# B&R Automation Studio project NAEUL004C00R13L518F00 (part 40)

### Buffer1.var - not listed in the package file held
```iecst
(*2019-06-07*)
(**)
(*Action & State & Status*)
VAR
	p_Buffer1Stat : UDINT;
	p_Buffer1Status : UDINT;
	p_Buffer1StatTxt : UDINT;
END_VAR
(**)
(*Alarm*)
VAR
	p_Buffer1AlmData : UDINT;
END_VAR
(**)
(*Output*)
VAR
	p_Buffer1NxtLoadSlt : UDINT;
	p_Buffer1NxtUnloadSlt : UDINT;
	p_Buffer1CoolBrdAny : UDINT;
	p_Buffer1CoolBrdGd : UDINT;
	p_Buffer1CoolBrdBad : UDINT;
	p_Buffer1CoolNotRdy : UDINT;
	p_Buffer1Bffr : UDINT;
	p_Buffer1DispBffr : UDINT;
	p_Buffer1BffrStat : UDINT;
	p_Buffer1BrdUnloadStat : UDINT;
	p_Buffer1FileNotFound : UDINT;
	p_Buffer1CoolFanCtrl : UDINT;
	p_Buffer1MagPresent : UDINT;
	p_Buffer1MagPresentTm : UDINT;
	p_Buffer1NewProduct : UDINT;
	p_Buffer1LastProductUnload : UDINT;
	p_Buffer1LastProductLeftInBffr : UDINT;
	p_Buffer1ParamDiff : UDINT;
	p_Buffer1MagRemoved : UDINT;
	p_Buffer1FIFOOld : UDINT;
	p_Buffer1SlotNo : UDINT;
END_VAR
```

### Buffer2.var - not listed in the package file held
```iecst
(*2019-03-25*)
(**)
(*Action & State & Status*)
VAR
	p_Buffer2Stat : UDINT;
	p_Buffer2Status : UDINT;
	p_Buffer2StatTxt : UDINT;
END_VAR
(**)
(*Alarm*)
VAR
	p_Buffer2AlmData : UDINT;
END_VAR
(**)
(*Output*)
VAR
	p_Buffer2NxtLoadSlt : UDINT;
	p_Buffer2NxtUnloadSlt : UDINT;
	p_Buffer2CoolBrdAny : UDINT;
	p_Buffer2CoolBrdGd : UDINT;
	p_Buffer2CoolBrdBad : UDINT;
	p_Buffer2CoolNotRdy : UDINT;
	p_Buffer2Bffr : UDINT;
	p_Buffer2DispBffr : UDINT;
	p_Buffer2BffrStat : UDINT;
	p_Buffer2BrdUnloadStat : UDINT;
	p_Buffer2FileNotFound : UDINT;
	p_Buffer2CoolFanCtrl : UDINT;
	p_Buffer2MagPresent : UDINT;
	p_Buffer2MagPresentTm : UDINT;
	p_Buffer2NewProduct : UDINT;
	p_Buffer2LastProductUnload : UDINT;
	p_Buffer2LastProductLeftInBffr : UDINT;
	p_Buffer2ParamDiff : UDINT;
	p_Buffer2MagRemoved : UDINT;
	p_Buffer2FIFOOld : UDINT;
	p_Buffer2SlotNo : UDINT;
END_VAR
```

### Buffer3.var - not listed in the package file held
```iecst
(*2019-03-25*)
(**)
(*Action & State & Status*)
VAR
	p_Buffer3Stat : UDINT;
	p_Buffer3Status : UDINT;
	p_Buffer3StatTxt : UDINT;
END_VAR
(**)
(*Alarm*)
VAR
	p_Buffer3AlmData : UDINT;
END_VAR
(**)
(*Output*)
VAR
	p_Buffer3NxtLoadSlt : UDINT;
	p_Buffer3NxtUnloadSlt : UDINT;
	p_Buffer3CoolBrdAny : UDINT;
	p_Buffer3CoolBrdGd : UDINT;
	p_Buffer3CoolBrdBad : UDINT;
	p_Buffer3CoolNotRdy : UDINT;
	p_Buffer3Bffr : UDINT;
	p_Buffer3DispBffr : UDINT;
	p_Buffer3BffrStat : UDINT;
	p_Buffer3BrdUnloadStat : UDINT;
	p_Buffer3FileNotFound : UDINT;
	p_Buffer3CoolFanCtrl : UDINT;
	p_Buffer3MagPresent : UDINT;
	p_Buffer3MagPresentTm : UDINT;
	p_Buffer3NewProduct : UDINT;
	p_Buffer3LastProductUnload : UDINT;
	p_Buffer3LastProductLeftInBffr : UDINT;
	p_Buffer3ParamDiff : UDINT;
	p_Buffer3MagRemoved : UDINT;
	p_Buffer3FIFOOld : UDINT;
	p_Buffer3SlotNo : UDINT;
END_VAR
```

### BufferMagA.var - not listed in the package file held
```iecst
(*2019-01-30*)
(**)
(*Action & State & Status*)
(**)
(*Alarm*)
(**)
(*Output*)
VAR
	p_BufferMagABffrMtySlt : UDINT;
END_VAR
```

### BufferMagB.var - not listed in the package file held
```iecst
(*2019-01-30*)
(**)
(*Action & State & Status*)
(**)
(*Alarm*)
(**)
(*Output*)
VAR
	p_BufferMagBBffrMtySlt : UDINT;
END_VAR
```

### SMEMA.typ - Do Not Change!!!
```iecst
(*2018-12-13*)
(**)
(*Action*)

TYPE
	eSMEMAAction :
		(
		SMEMAActIdle,
		SMEMAActRun,
		SMEMAActSetSig,
		SMEMAActSetStatSig,
		SMEMAActRstSig,
		SMEMAActRstStatSig,
		SMEMAActSetAllSig,
		SMEMAActRstAllSig
		);
END_TYPE

(**)

TYPE
	tySMEMAParam : 	STRUCT
		eSelection : eSMEMASelection;
		bStatSigSetGd : BOOL;
	END_STRUCT;
	eSMEMASelection :
		(
		SMEMASelStandard,
		SMEMASelIPC9851,
		SMEMASelIPC9851Ext
		);
	tyUSSMEMA : 	STRUCT
		In : tyUSSMEMAIn1;
		Out : tyUSSMEMAAOut1;
	END_STRUCT;
	tyUSSMEMAIn1 : 	STRUCT
		eAct : eSMEMAAction := SMEMAActIdle; (*USSMEMA Act*)
		udiRstErr : UDINT := 0; (*Reset Error*)
		bPrep : BOOL := TRUE; (*Project Preparation*)
		bEn : BOOL := TRUE; (*Enable*)
		bDis : BOOL := FALSE; (*Disable*)
		bRdyRcv : BOOL := TRUE; (*Ready Receive Signal*)
		bLeftSen : BOOL := FALSE; (*Left Sensor*)
		bRightSen : BOOL := FALSE; (*Right Sensor*)
		bComplSigOn : BOOL := FALSE; (*Complete Signal is On*)
		bUBA : BOOL := FALSE; (*Upstream is Available Signal*)
		bUBAStat : BOOL := FALSE; (*Upstream is Available Signal's State*)
		bTimerEnSen : BOOL; (*Timer Enable Sensor*)
		bTimerEnSenEdge : BOOL; (*Timer Enable Sensor Edge*)
		bVirtualEn : BOOL; (*Virtual Mode Enable*)
		bUBAVirtual : BOOL; (*Upstream Available Vritual Signal*)
		bUBAStatVirtual : BOOL; (*Upstream Available Vritual Signal's State*)
		tyParam : tySMEMAParam; (*SMEMA Parameter*)
		diTransferInTO : DINT := 20000; (*Transfer Out Timer On*)
		bDirLToR : BOOL := FALSE; (*Direction Left to Right*)
		tRstDlyTm : TIME := T#500ms; (*Reset Delay Timer*)
		tSigInChkTm : TIME := T#100ms; (*Signal In Check Timer*)
		sProgNm : STRING[15] := 'USSMEMA'; (*Program's Name*)
		bNtSettingsLoadDone : BOOL := TRUE; (*Nutek Parameter Settings Loading is Done*)
	END_STRUCT;
	tyUSSMEMAAOut1 : 	STRUCT
		eStat : eBufferAction := BufferActIdle; (*Hardware Info's State*)
		eStatus : eFBStatus := Idle; (*Hardware Info's Status*)
		sStatTxt : STRING[200] := ''; (*Hardware Info's State in Text*)
		tyAlmData : tyAlmDat; (*Alarm Data*)
		bUSRdy : BOOL := FALSE; (*Upstream is Ready*)
		bUSGdBrdRdy : BOOL := FALSE; (*Upstream Good Board is Ready*)
		bDSRdy : BOOL := FALSE; (*Downstream is Ready*)
		bTransporting : BOOL := FALSE; (*Is Transporting*)
		bConvStart : BOOL := FALSE; (*Converyor Starts*)
		bConvStop : BOOL := FALSE; (*Conveyor Stop*)
		bUSB : BOOL := FALSE; (*Upstream Busy Signal*)
		bTimer : BOOL; (*Timer is On*)
		bVirtual : BOOL; (*Virtual Mode is On*)
	END_STRUCT;
	tyDSSMEMA : 	STRUCT
		In : tyDSSMEMAIn1;
		Out : tyDSSMEMAOut1;
	END_STRUCT;
	tyDSSMEMAIn1 : 	STRUCT
		eAct : eSMEMAAction := SMEMAActIdle; (*DSSMEMA Act*)
		udiRstErr : UDINT := 0; (*Reset Error*)
		bPrep : BOOL := TRUE; (*Project Preparation*)
		bEn : BOOL := TRUE; (*Enable*)
		bDis : BOOL := FALSE; (*Disable*)
		bGdBrd : BOOL := TRUE; (*Have Good Board*)
		bRdySend : BOOL := TRUE; (*Ready Send Signal*)
		bLeftSen : BOOL := FALSE; (*Left Sensor*)
		bRightSen : BOOL := FALSE; (*Right Sensor*)
		bClrSen : BOOL;
		bComplSigOn : BOOL := FALSE; (*Complete Signal is On*)
		bDSB : BOOL := FALSE; (*Downstream Busy Signal*)
		bTimerEnSen : BOOL; (*Timer Enable Sensor*)
		bTimerEnSenEdge : BOOL; (*Timer Enable Sensor Edge*)
		bVirtualEn : BOOL; (*Virtual Mode Enable*)
		bDSBVirtual : BOOL; (*Downstream Busy Signal*)
		tyParam : tySMEMAParam; (*SMEMA Parameter*)
		diTransferOutTO : DINT := 20000;
		bDirLToR : BOOL := FALSE; (*Direction Left to Right*)
		tRstDlyTm : TIME := T#500ms; (*Reset Delay Timer*)
		tSigInChkTm : TIME := T#100ms; (*Signal In Check Timer*)
		sProgNm : STRING[15] := 'USSMEMA'; (*Program's Name*)
		bNtSettingsLoadDone : BOOL := TRUE; (*Nutek Parameter Settings Loading is Done*)
	END_STRUCT;
	tyDSSMEMAOut1 : 	STRUCT
		eStat : eSMEMAAction := SMEMAActIdle; (*DSSMEMA's State*)
		eStatus : eFBStatus := Idle; (*DSSMEMA's Status*)
		sStatTxt : STRING[200] := ''; (*DSSMEMA's State in Text*)
		tyAlmData : tyAlmDat; (*Alarm Data*)
		bUSRdy : BOOL := FALSE; (*Upstream is Ready*)
		bUSGdBrdRdy : BOOL := FALSE; (*Upstream Good Board is Ready*)
		bDSRdy : BOOL := FALSE; (*Downstream is Ready*)
		bTransporting : BOOL := FALSE; (*Is Transporting*)
		bConvStart : BOOL := FALSE; (*Conveyor Start*)
		bConvStop : BOOL := FALSE; (*Conveyor Stop*)
		bDBA : BOOL := FALSE; (*Downstream Available Signal*)
		bDBAStat : BOOL := FALSE; (*Downstream Avaialble Signal's State*)
		bTimer : BOOL; (*Timer is On*)
		bVirtual : BOOL; (*Virtual Mode is Mode*)
	END_STRUCT;
END_TYPE
```

### USSMEMAA.var - Change By Project
```iecst
(**)
VAR
	g_tyUSSMEMAA : tyUSSMEMAAOut1; (*Upstream SMEMA*)
END_VAR
```

### Program Logical/SMEMA/USSMEMAA (IEC) - 1.00.0 - NtSMEMA v5.00.0

#### InputRef_Link.var
```iecst
(*2019-04-09*)
(**)
(*External Data*)
VAR
	p_bLinkOpsRun : REFERENCE TO BOOL;
END_VAR
(**)
VAR
	p_eLinkConvDir : REFERENCE TO eConvDir;
	p_eLinkOpsTravLifPosGo : REFERENCE TO eTravLifULPos;
	p_bLinkConvHvBrd : REFERENCE TO BOOL;
	p_bLinkNtParamUSWidthChkPrep : REFERENCE TO BOOL;
	p_bLinkMcParamUSWidthChkEn : REFERENCE TO BOOL;
	p_bLinkDIUSWidthChkSen : REFERENCE TO BOOL;
END_VAR
```

#### Act_Alarm.st
```iecst
(** 2019-03-25 **)
ACTION Act_Alarm:
	//Reset Error
	IF tylocalUSSMEMA.In.udiRstErr <> udiRstErrOld THEN
		bRstErr			:= TRUE;
		udiRstErrOld	:= tylocalUSSMEMA.In.udiRstErr;
	ELSE
		bRstErr			:= FALSE;
	END_IF

	//Error State
	IF (tylocalUSSMEMA.Out.eStatus = Error) AND bRstErr THEN
		tylocalUSSMEMA.In.eAct		:= SMEMAActIdle;
		tylocalUSSMEMA.Out.eStat	:= SMEMAActIdle;
	END_IF

	//Error Link To HMI
	IF EDGEPOS(tylocalUSSMEMA.Out.eStatus = Error) THEN

		tylocalUSSMEMA.Out.tyAlmData.udiCode		:= udiStatus;
		tylocalUSSMEMA.Out.tyAlmData.eSeverity		:= AlmSeverityError;
		tylocalUSSMEMA.Out.tyAlmData.udiRunTime		:= tylocalUSSMEMA.Out.tyAlmData.udiRunTime + 1;
		tylocalUSSMEMA.Out.tyAlmData.bAlm			:= TRUE;
		tylocalUSSMEMA.Out.tyAlmData.udiModuleNum	:= udiModuleNum;
		g_tyAlmProgNm.sUSSMEMAProgNm				:= tylocalUSSMEMA.In.sProgNm;

	ELSIF bRstErr AND (tylocalUSSMEMA.Out.tyAlmData.udiCode <> 0) THEN

		tylocalUSSMEMA.Out.tyAlmData.udiCode	:= 0;
		tylocalUSSMEMA.Out.tyAlmData.eSeverity	:= AlmSeverityNA;
		tylocalUSSMEMA.Out.tyAlmData.bAlm		:= FALSE;

		tylocalUSSMEMA.Out.sStatTxt	:= a_sStatText[tylocalUSSMEMA.Out.eStat];

	END_IF

END_ACTION
```

#### Act_InitGlobal.st
```iecst
(** 2019-04-09 **)
ACTION Act_InitGlobal:

	(* Always Change If Project Change *)

	//Pass Data To Link
	p_bLinkOpsRun ACCESS p_OpsRun;

	p_eLinkConvDir ACCESS p_NtParamProjConvDir;
	p_eLinkOpsTravLifPosGo ACCESS p_OpsTravLifULPosGo;
	p_bLinkConvHvBrd ACCESS p_PshrConvHvBrd;
	p_bLinkNtParamUSWidthChkPrep ACCESS p_NtParamUSWidthChkPrep;
	p_bLinkMcParamUSWidthChkEn ACCESS p_McParamUSWidthChkEn;
	p_bLinkDIUSWidthChkSen ACCESS p_DIUSWidthChkSen;

	//Pass Data To Internal Use
	p_udiRstErr ACCESS p_RstErrReset;
	p_bManual ACCESS p_UIMnlMod;
	p_tyParam ACCESS p_McParamUSSMEMAAParam;
	p_diTransferInTO ACCESS p_McParamTranInErrDlyTm;
	p_bLeftSen ACCESS p_DIConvLftSen;
	p_bRightSen ACCESS p_DIConvRgtSen;
	p_bUBA ACCESS p_DIUBAA;
	p_bUBAStat ACCESS p_DIUBAAStat;
	p_bVirtualEn ACCESS p_UIVSMEMAUSAEn;
	p_bUBAVirtual ACCESS p_UIVSMEMAUBAA;
	p_bUBAStatVirtual ACCESS p_UIVSMEMAUBAAStat;
	p_tRstDlyTm ACCESS p_NtParamUSSMEMAARstDlyTm;
	p_tSigInChkTm ACCESS p_NtParamUSSMEMAASigInChkTm;
	p_sProgNm ACCESS p_NtParamUSSMEMAAProgNm;
	p_bNtSettingsLoadDone ACCESS p_StartupNtSettingsLoadDone;
	p_bLinkOpsTravLifULUSComm ACCESS p_OpsTravLifULUSComm;
	(* Always Change If Project Change *)

END_ACTION
```

#### Act_InputConfig.st
```iecst
(** 2019-04-09 **)
ACTION Act_InputConfig:

	(* Always Change If Project Change *)

	//Pass Data To Link
	tylocalUSSMEMA.In.udiRstErr := g_tyRstErr.bReset;
	tylocalUSSMEMA.In.tyParam := g_tyMcParamCurr.tyUSCommASMEMA;
	tylocalUSSMEMA.In.diTransferInTO := g_tyMcParamCurr.diTranInErrDlyTmInMS;
	tylocalUSSMEMA.In.bLeftSen := g_tyDInput.bConvLftSen;
	tylocalUSSMEMA.In.bRightSen := g_tyDInput.bConvRgtSen;
	tylocalUSSMEMA.In.bUBA := g_tyDInput.bUBAA;
	tylocalUSSMEMA.In.bUBAStat := g_tyDInput.bUBAAStat;
	tylocalUSSMEMA.In.bVirtualEn := g_tyUIOut.bVSMEMAUSAEn;
	tylocalUSSMEMA.In.bUBAVirtual := g_tyUIOut.bVSMEMAUBAA;
	tylocalUSSMEMA.In.bUBAStatVirtual := g_tyUIOut.bVSMEMAUBAAStat;
	tylocalUSSMEMA.In.tRstDlyTm := g_tyNtParamCurr.tUSSMEMAARstDlyTm;
	tylocalUSSMEMA.In.tSigInChkTm := g_tyNtParamCurrt.tUSSMEMAASigInChkTm;
	tylocalUSSMEMA.In.sProgNm := g_tyNtParamCurr.sUSSMEMAAProgNm;

	//Ready Receive
	IF g_tyNtParamCurr.bUSWidthChkPrep AND g_tyMcParamCurr.bUSWidthChkEn THEN
		tylocalUSSMEMA.In.bRdyRcv	:= (g_tyDInput.bnput.bUSWidthChkSen = TRUE) AND (g_tyPshrConv.bHvBrd = FALSE) AND (g_tyOpsTravLifUL.eTravLifULPosGo = TravLifULPosUS1);
	ELSE
		tylocalUSSMEMA.In.bRdyRcv	:= (g_tyPshrConv.bHvBrd = FALSE) AND (g_tyOpsTravLifUL.eTravLifULPosGo = TravLifULPosUS1) AND g_tyOps.bTravLifULUSComm;
	END_IF

	//Receive Complete Signal
	//	tylocalUSSMEMA.In.bComplSigOn	:= tylocalUSSMEMA.In.bLeftSen = FALSE;
	IF EDGENEG(tylocalUSSMEMA.In.bLeftSen) THEN
		tylocalUSSMEMA.In.bComplSigOn	:= TRUE;
	END_IF

	IF tylocalUSSMEMA.Out.eStat <> SMEMAActRun THEN
		tylocalUSSMEMA.In.bComplSigOn	:= FALSE;
	END_IF

	//Direction
	tylocalUSSMEMA.In.bDirLToR	:= g_tyNtParamCurr.eProjConvDir = ConvDirLToR OR g_tyNtParamCurr.eProjConvDir = ConvDirRToL;

	IF g_tyOps.bRun = TRUE THEN
		tylocalUSSMEMA.In.eAct := g_tyOpsTravLifUL.eUSSMEMAAct1;
	ELSIF g_tyUIOut.Out.bManualMod = TRUE THEN
		tylocalUSSMEMA.In.eAct := g_tyUIOut.eMnlAct.eUSSMEMAAAct;
	ELSE
		tylocalUSSMEMA.In.eAct ACCESS ADR(eAct);
	END_IF

END_ACTION
```

#### Act_Link.st
```iecst
(** 2019-03-29 **)
ACTION Act_Link:

	//Ready Receive
	IF p_bLinkNtParamUSWidthChkPrep AND p_bLinkMcParamUSWidthChkEn THEN
		p_bRdyRcv	:= (p_bLinkDIUSWidthChkSen = TRUE) AND (p_bLinkConvHvBrd = FALSE) AND (p_eLinkOpsTravLifPosGo = TravLifULPosUS1);
	ELSE
		p_bRdyRcv	:= (p_bLinkConvHvBrd = FALSE) AND (p_eLinkOpsTravLifPosGo = TravLifULPosUS1) AND p_bLinkOpsTravLifULUSComm;
	END_IF

	//Receive Complete Signal
//	p_bComplSigOn	:= p_bLeftSen = FALSE;
	IF EDGENEG(p_bLeftSen) THEN
		p_bComplSigOn	:= TRUE;
	END_IF

	IF eStat <> SMEMAActRun THEN
		p_bComplSigOn	:= FALSE;
	END_IF

	//Direction
	p_bDirLToR	:= p_eLinkConvDir = ConvDirLToR OR p_eLinkConvDir = ConvDirLToL;

END_ACTION
```

#### Act_LinkAction.st
```iecst
(** 2019-04-09 **)
ACTION Act_LinkAction:

	IF p_bLinkOpsRun = TRUE THEN
		p_eAct ACCESS p_OpsTravLifULUSSMEMAAct1;
	ELSIF p_bManual = TRUE THEN
		p_eAct ACCESS p_UIUSSMEMAAAct;
	ELSE
		p_eAct ACCESS ADR(eAct);
	END_IF

END_ACTION
```

#### Act_Main.st
```iecst
ACTION Act_Main:

	fbSMEMA_Std.tRstDlyTm 		:= tylocalUSSMEMA.In.tRstDlyTm;
	fbSMEMA_9851.tRstDlyTm  	:= tylocalUSSMEMA.In.tRstDlyTm;
	fbSigInChk.tSigInChkTm		:= tylocalUSSMEMA.In.tSigInChkTm;

	//Timer Running
	fbTimeTrig(CLK := tylocalUSSMEMA.In.bTimerEnSenEdge);

	IF tylocalUSSMEMA.Out.eStat = SMEMAActRun AND (tylocalUSSMEMA.In.bTimerEnSenEdge OR tylocalUSSMEMA.In.bTimerEnSen) THEN
		IF fbTimeTrig.Q = TRUE OR tylocalUSSMEMA.In.bTimerEnSen THEN
			fbTimerDlyTm.IN	:= TRUE;
		END_IF
	ELSE
		fbTimerDlyTm.IN	:= FALSE;
	END_IF

	IF tylocalUSSMEMA.Out.bConvStart = FALSE AND tylocalUSSMEMA.Out.bConvStop = FALSE THEN
		fbTimerDlyTm;

		IF fbTimerDlyTm.Q = TRUE AND tylocalUSSMEMA.Out.eStat = SMEMAActRun THEN
			tylocalUSSMEMA.Out.bTimer		:= TRUE;
			tylocalUSSMEMA.Out.bVirtual		:= FALSE;
		ELSIF tylocalUSSMEMA.In.bVirtualEn = TRUE THEN
			tylocalUSSMEMA.Out.bTimer		:= FALSE;
			tylocalUSSMEMA.Out.bVirtual		:= TRUE;
		ELSE
			tylocalUSSMEMA.Out.bTimer		:= FALSE;
			tylocalUSSMEMA.Out.bVirtual		:= FALSE;
		END_IF
	ELSE
		fbTimerDlyTm(IN := FALSE);
	END_IF

	IF tylocalUSSMEMA.Out.bTimer = TRUE THEN

		fbSigInChk.bNomSig			:= tylocalUSSMEMA.Out.bConvStart = FALSE AND tylocalUSSMEMA.Out.bConvStop = FALSE;
		fbSigInChk.bStatSig			:= FALSE;
		fbSigInChk.bStatSigSetGd	:= FALSE;

	ELSIF tylocalUSSMEMA.Out.bVirtual = TRUE THEN

		fbSigInChk.bNomSig	:= tylocalUSSMEMA.In.bUBAVirtual;

		IF tylocalUSSMEMA.In.tyParam.eSelection = SMEMASelIPC9851Ext THEN
			fbSigInChk.bStatSig			:= tylocalUSSMEMA.In.bUBAStatVirtual;
			fbSigInChk.bStatSigSetGd	:= tylocalUSSMEMA.In.tyParam.bStatSigSetGd;
		ELSE
			fbSigInChk.bStatSig			:= FALSE;
			fbSigInChk.bStatSigSetGd	:= FALSE;
		END_IF

	ELSE

		fbSigInChk.bNomSig	:= tylocalUSSMEMA.In.bUBA;

		IF tylocalUSSMEMA.In.tyParam.eSelection = SMEMASelIPC9851Ext THEN
			fbSigInChk.bStatSig			:= tylocalUSSMEMA.In.bUBAStat;
			fbSigInChk.bStatSigSetGd	:= tylocalUSSMEMA.In.tyParam.bStatSigSetGd;
		ELSE
			fbSigInChk.bStatSig			:= FALSE;
			fbSigInChk.bStatSigSetGd	:= FALSE;
		END_IF

	END_IF

	fbSigInChk;

	tylocalUSSMEMA.Out.bUSRdy		    := fbSigInChk.bSigInValid;
	tylocalUSSMEMA.Out.bUSGdBrdRdy   	:= fbSigInChk.bGdBrd;

	//Set p_eAct
	IF tylocalUSSMEMA.Out.eStatus = Idle OR tylocalUSSMEMA.Out.eStatus = Busy OR tylocalUSSMEMA.Out.eStatus = Done THEN
		tylocalUSSMEMA.Out.eStatus	:= tylocalUSSMEMA.In.eAct;
	END_IF

	//Transition State
	IF eStatOld <> tylocalUSSMEMA.Out.eStat THEN

		fbSMEMA_Std(bEn := FALSE);
		fbSMEMA_9851(bEn := FALSE);

		tylocalUSSMEMA.Out.bTransporting	:= FALSE;
		tylocalUSSMEMA.Out.bConvStart		:= FALSE;
		tylocalUSSMEMA.Out.bConvStop		:= FALSE;
		tylocalUSSMEMA.Out.bDSRdy			:= FALSE;

		IF eStatOld <> SMEMAActIdle
			AND eStatOld <> SMEMAActSetSig
			AND eStatOld <> SMEMAActSetStatSig
			AND eStatOld <> SMEMAActRstSig
			AND eStatOld <> SMEMAActRstStatSig
			AND eStatOld <> SMEMAActSetAllSig
			AND eStatOld <> SMEMAActRstAllSig THEN

			tylocalUSSMEMA.Out.bUSB	:= FALSE;

		END_IF

		tylocalUSSMEMA.Out.sStatTxt	:= a_sStatText[tylocalUSSMEMA.Out.eStat];

		eStatOld	:= tylocalUSSMEMA.Out.eStat;

		tylocalUSSMEMA.Out.eStatus		:= Busy;
	END_IF

	//Inlet Sensor & Outlet Sensor
	IF tylocalUSSMEMA.In.bDirLToR THEN
		bInletSen 	:= tylocalUSSMEMA.In.bLeftSen;
		bOutletSen  := tylocalUSSMEMA.In.bRightSen;
	ELSE
		bInletSen   := tylocalUSSMEMA.In.bRightSen;
		bOutletSen  := tylocalUSSMEMA.In.bLeftSen;
	END_IF

	//Main
	CASE tylocalUSSMEMA.Out.eStat OF

		SMEMAActIdle:

			IF EDGENEG(g_tyUIOut.bManualMod) THEN
				tylocalUSSMEMA.Out.bUSB	:= FALSE;
			END_IF

			tylocalUSSMEMA.Out.eStatus	:= Idle;

		SMEMAActRun:
			IF tylocalUSSMEMA.Out.eStatus = Idle OR tylocalUSSMEMA.Out.eStatus = Busy THEN

				tylocalUSSMEMA.Out.eStatus	:= Busy;

				IF tylocalUSSMEMA.In.tyParam.eSelection <> SMEMASelStandard THEN

					fbSMEMA_9851.bUSRdy			:= fbSigInChk.bSigInValid;
					fbSMEMA_9851.bRdyRcv		:= tylocalUSSMEMA.In.bRdyRcv;
					fbSMEMA_9851.bComplSigOn	:= tylocalUSSMEMA.In.bComplSigOn;
					fbSMEMA_9851.bInletSen		:= bInletSen;
					fbSMEMA_9851.bOutletSen		:= bOutletSen;

					fbSMEMA_9851.tTimeOut		:= DINT_TO_TIME(tylocalUSSMEMA.In.diTransferInTO);
					fbSMEMA_9851(bEn := TRUE);

					tylocalUSSMEMA.Out.bTransporting	:= fbSMEMA_9851.bTransporting;
					tylocalUSSMEMA.Out.bConvStart		:= fbSMEMA_9851.bConvStart;
					tylocalUSSMEMA.Out.bConvStop		:= fbSMEMA_9851.bConvStop;
					tylocalUSSMEMA.Out.bUSB				:= fbSMEMA_9851.bSigToUS AND (tylocalUSSMEMA.Out.bTimer = FALSE) AND (tylocalUSSMEMA.Out.bVirtual = FALSE);
					tylocalUSSMEMA.Out.bDSRdy			:= fbSMEMA_9851.bSigToUS;

					IF fbSMEMA_9851.udiStatus = 0 THEN
						tylocalUSSMEMA.Out.eStatus	:= Done;
					ELSIF fbSMEMA_9851.udiStatus < 65534 THEN
						tylocalUSSMEMA.Out.eStatus		:= Error;

						IF fbSMEMA_9851.udiStatus = 1200 THEN
							udiStatus	:= 2701;	//SMEMA 9851 Transport Time Out While Transporting
						ELSIF fbSMEMA_9851.udiStatus = 1201 THEN
							udiStatus	:= 2702;	//SMEMA 9851 Transport Time Out After Opposite Machine Transport Finished
						ELSIF fbSMEMA_9851.udiStatus = 1202 THEN
							udiStatus	:= 2703;	//SMEMA 9851 Transport Time Out After Current Machine Transport Finished
						ELSIF fbSMEMA_9851.udiStatus = 1203 THEN
							udiStatus	:= 2704;	//SMEMA 9851 Transport Time Out After Both Machine Transport Finished And Waiting Outlet Sensor
						ELSE
							udiStatus	:= fbSMEMA_9851.udiStatus;
						END_IF
					END_IF

				ELSE

					fbSMEMA_Std.bUSRdy		:= fbSigInChk.bSigInValid;
					fbSMEMA_Std.bRdyRcv		:= tylocalUSSMEMA.In.bRdyRcv;
					fbSMEMA_Std.bComplSigOn	:= tylocalUSSMEMA.In.bComplSigOn;
					fbSMEMA_Std.bInletSen	:= bInletSen;
					fbSMEMA_Std.bOutletSen	:= bOutletSen;
					fbSMEMA_Std.tTimeOut	:= DINT_TO_TIME(tylocalUSSMEMA.In.diTransferInTO);
					fbSMEMA_Std(bEn := TRUE);

					tylocalUSSMEMA.Out.bTransporting	:= fbSMEMA_Std.bTransporting;
					tylocalUSSMEMA.Out.bConvStart		:= fbSMEMA_Std.bConvStart;
					tylocalUSSMEMA.Out.bConvStop		:= fbSMEMA_Std.bConvStop;
					tylocalUSSMEMA.Out.bUSB				:= fbSMEMA_Std.bSigToUS AND (tylocalUSSMEMA.Out.bTimer = FALSE) AND (tylocalUSSMEMA.Out.bVirtual = FALSE);
					tylocalUSSMEMA.Out.bDSRdy			:= fbSMEMA_Std.bSigToUS;

					IF fbSMEMA_Std.udiStatus = 0 THEN
						tylocalUSSMEMA.Out.eStatus	:= Done;
					ELSIF fbSMEMA_Std.udiStatus < 65534 THEN
						tylocalUSSMEMA.Out.eStatus		:= Error;

						IF fbSMEMA_Std.udiStatus = 1200 THEN
							udiStatus	:= 2705;	//Standard SMEMA Transport Time Out While Transporting
						ELSIF fbSMEMA_Std.udiStatus = 1201 THEN
							udiStatus	:= 2706;	//Standard SMEMA Transport Time Out After Opposite Machine Transport Finished
						ELSIF fbSMEMA_Std.udiStatus = 1202 THEN
							udiStatus	:= 2707;	//Standard SMEMA Transport Time Out After Current Machine Transport Finished
						ELSIF fbSMEMA_Std.udiStatus = 1203 THEN
							udiStatus	:= 2708;	//Standard SMEMA Transport Time Out After Both Machine Transport Finished And Waiting Outlet Sensor
						ELSE
							udiStatus	:= fbSMEMA_Std.udiStatus;
						END_IF
					END_IF

				END_IF

			END_IF

		SMEMAActSetSig:
			IF tylocalUSSMEMA.Out.eStatus = Idle OR tylocalUSSMEMA.Out.eStatus = Busy THEN

				//Reset
				fbSMEMA_Std(bEn := FALSE);
				fbSMEMA_9851(bEn := FALSE);

				tylocalUSSMEMA.Out.bConvStart	:= FALSE;
				tylocalUSSMEMA.Out.bConvStop	:= FALSE;

				tylocalUSSMEMA.Out.bUSB		:= TRUE;
				tylocalUSSMEMA.Out.eStatus	:= Done;

			END_IF

		SMEMAActSetStatSig:
			IF tylocalUSSMEMA.Out.eStatus = Idle OR tylocalUSSMEMA.Out.eStatus = Busy THEN

				//Reset
				fbSMEMA_Std(bEn := FALSE);
				fbSMEMA_9851(bEn := FALSE);

				tylocalUSSMEMA.Out.bConvStart	:= FALSE;
				tylocalUSSMEMA.Out.bConvStop	:= FALSE;

				tylocalUSSMEMA.Out.eStatus	:= Done;

			END_IF

		SMEMAActRstSig:
			IF tylocalUSSMEMA.Out.eStatus = Idle OR tylocalUSSMEMA.Out.eStatus = Busy THEN

				//Reset
				fbSMEMA_Std(bEn := FALSE);
				fbSMEMA_9851(bEn := FALSE);

				tylocalUSSMEMA.Out.bConvStart	:= FALSE;
				tylocalUSSMEMA.Out.bConvStop	:= FALSE;

				tylocalUSSMEMA.Out.bUSB	:= FALSE;
				tylocalUSSMEMA.Out.eStatus	:= Done;

			END_IF

		SMEMAActRstStatSig:
			IF tylocalUSSMEMA.Out.eStatus = Idle OR tylocalUSSMEMA.Out.eStatus = Busy THEN

				//Reset
				fbSMEMA_Std(bEn := FALSE);
				fbSMEMA_9851(bEn := FALSE);

				tylocalUSSMEMA.Out.bConvStart	:= FALSE;
				tylocalUSSMEMA.Out.bConvStop	:= FALSE;

				tylocalUSSMEMA.Out.eStatus	:= Done;

			END_IF

		SMEMAActSetAllSig:
			IF tylocalUSSMEMA.Out.eStatus = Idle OR tylocalUSSMEMA.Out.eStatus = Busy THEN

				//Reset
				fbSMEMA_Std(bEn := FALSE);
				fbSMEMA_9851(bEn := FALSE);

				tylocalUSSMEMA.Out.bConvStart	:= FALSE;
				tylocalUSSMEMA.Out.bConvStop	:= FALSE;

				tylocalUSSMEMA.Out.bUSB	:= TRUE;
				tylocalUSSMEMA.Out.eStatus	:= Done;

			END_IF

		SMEMAActRstAllSig:
			IF tylocalUSSMEMA.Out.eStatus = Idle OR tylocalUSSMEMA.Out.eStatus = Busy THEN

				//Reset
				fbSMEMA_Std(bEn := FALSE);
				fbSMEMA_9851(bEn := FALSE);

				tylocalUSSMEMA.Out.bConvStart	:= FALSE;
				tylocalUSSMEMA.Out.bConvStop	:= FALSE;

				tylocalUSSMEMA.Out.bUSB	:= FALSE;
				tylocalUSSMEMA.Out.eStatus	:= Done;

			END_IF

	END_CASE

END_ACTION
```

#### Act_OutputConfig.st
```iecst
(** 2019-03-25 **)
ACTION Act_OutputConfig:

	g_tyUSSMEMAA := tylocalUSSMEMA.Out; // Change the Global Naming According to the Physical Hardware Module

END_ACTION
```

#### Init.st
```iecst
(** 2019-03-25 **)
PROGRAM _INIT

	(* Always Change If Project Change *)

	//Pass Address To Global Address For External Use
	//Action, State & Status
	p_USSMEMAAStat		:= ADR(eStat);
	p_USSMEMAAStatus		:= ADR(eStatus);
	p_USSMEMAAStatTxt	:= ADR(sStatTxt);

	//Alarm
	p_USSMEMAAAlmData	:= ADR(tyAlmData);

	//Output
	p_USSMEMAAUSRdy			:= ADR(bUSRdy);
	p_USSMEMAAUSGdBrdRdy	:= ADR(bUSGdBrdRdy);
	p_USSMEMAADSRdy			:= ADR(bDSRdy);
	p_USSMEMAATransporting	:= ADR(bTransporting);
	p_USSMEMAAConvStart		:= ADR(bConvStart);
	p_USSMEMAAConvStop		:= ADR(bConvStop);
	p_USSMEMAAUSB			:= ADR(bUSB);
	p_USSMEMAATimer			:= ADR(bTimer);
	p_USSMEMAAVirtual		:= ADR(bVirtual);

	(* Always Change If Project Change *)

END_PROGRAM
```

### USSMEMAB.var - Change By Project
```iecst
VAR
	g_tyUSSMEMAB : tyUSSMEMAAOut1;
END_VAR
```

### Program Logical/SMEMA/USSMEMAB (IEC) - 1.00.0 - NtSMEMA v5.00.0

#### InputRef.var
```iecst
(*2019-03-25*)
(**)
(*General*)
VAR
	p_eAct : REFERENCE TO eSMEMAAction;
	p_udiRstErr : REFERENCE TO UDINT;
	p_bPrep : REFERENCE TO BOOL;
	p_bEn : REFERENCE TO BOOL;
	p_bDis : REFERENCE TO BOOL;
END_VAR
(**)
(*Configuration*)
VAR
	p_bManual : REFERENCE TO BOOL;
	p_tyParam : REFERENCE TO tySMEMAParam;
	p_diTransferInTO : REFERENCE TO DINT;
	p_bDirLToR : REFERENCE TO BOOL;
	p_bRdyRcv : REFERENCE TO BOOL;
END_VAR
(**)
(*Input*)
VAR
	p_bLeftSen : REFERENCE TO BOOL;
	p_bRightSen : REFERENCE TO BOOL;
	p_bComplSigOn : REFERENCE TO BOOL;
	p_bUBA : REFERENCE TO BOOL;
	p_bUBAStat : REFERENCE TO BOOL;
	p_bTimerEnSen : REFERENCE TO BOOL;
	p_bTimerEnSenEdge : REFERENCE TO BOOL;
	p_bVirtualEn : REFERENCE TO BOOL;
	p_bUBAVirtual : REFERENCE TO BOOL;
	p_bUBAStatVirtual : REFERENCE TO BOOL;
	p_tRstDlyTm : REFERENCE TO TIME;
	p_tSigInChkTm : REFERENCE TO TIME;
	p_sProgNm : REFERENCE TO STRING[15];
	p_bNtSettingsLoadDone : REFERENCE TO BOOL;
	p_bLinkOpsTravLifULUSComm : REFERENCE TO BOOL;
END_VAR
```

#### Act_InitGlobal.st
```iecst
(** 2019-04-09 **)
ACTION Act_InitGlobal:

	(* Always Change If Project Change *)

	//Pass Data To Link
	p_bLinkOpsRun ACCESS p_OpsRun;

	p_eLinkConvDir ACCESS p_NtParamProjConvDir;
	p_eLinkOpsTravLifPosGo ACCESS p_OpsTravLifULPosGo;
	p_bLinkConvHvBrd ACCESS p_PshrConvHvBrd;
	p_bLinkNtParamUSWidthChkPrep ACCESS p_NtParamUSWidthChkPrep;
	p_bLinkMcParamUSWidthChkEn ACCESS p_McParamUSWidthChkEn;
	p_bLinkDIUSWidthChkSen ACCESS p_DIUSWidthChkSen;

	//Pass Data To Internal Use
	p_udiRstErr ACCESS p_RstErrReset;
	p_bManual ACCESS p_UIMnlMod;
	p_tyParam ACCESS p_McParamUSSMEMABParam;
	p_diTransferInTO ACCESS p_McParamTranInErrDlyTm;
	p_bLeftSen ACCESS p_DIConvLftSen;
	p_bRightSen ACCESS p_DIConvRgtSen;
	p_bUBA ACCESS p_DIUBAB;
	p_bUBAStat ACCESS p_DIUBABStat;
	p_bVirtualEn ACCESS p_UIVSMEMAUSBEn;
	p_bUBAVirtual ACCESS p_UIVSMEMAUBAB;
	p_bUBAStatVirtual ACCESS p_UIVSMEMAUBABStat;
	p_tRstDlyTm ACCESS p_NtParamUSSMEMABRstDlyTm;
	p_tSigInChkTm ACCESS p_NtParamUSSMEMABSigInChkTm;
	p_sProgNm ACCESS p_NtParamUSSMEMABProgNm;
	p_bNtSettingsLoadDone ACCESS p_StartupNtSettingsLoadDone;
	p_bLinkOpsTravLifULUSComm ACCESS p_OpsTravLifULUSComm;
	(* Always Change If Project Change *)

END_ACTION
```

#### Act_Initial.st
```iecst
ACTION Act_Initial:

	//Initial
	tylocalUSSMEMA.Out.sStatTxt		:= a_sStatText[tylocalUSSMEMA.Out.eStat];
	fbSMEMA_Std(bEn := FALSE);
	fbSMEMA_9851(bEn := FALSE);
	fbTimerDlyTm(IN := FALSE);
	fbTimeTrig(CLK := TRUE);

END_ACTION
```

#### Act_InputConfig.st
```iecst
(** 2019-04-09 **)
ACTION Act_InputConfig:

	(* Always Change If Project Change *)

	//Pass Data To Link
	tylocalUSSMEMA.In.udiRstErr := g_tyRstErr.bReset;
	tylocalUSSMEMA.In.tyParam := g_tyMcParamCurr.tyUSCommBSMEMA;
	tylocalUSSMEMA.In.diTransferInTO := g_tyMcParamCurr.diTranInErrDlyTmInMS;
	tylocalUSSMEMA.In.bLeftSen := g_tyDInput.bConvLftSen;
	tylocalUSSMEMA.In.bRightSen := g_tyDInput.bConvRgtSen;
	tylocalUSSMEMA.In.bUBA := g_tyDInput.bUBAB;
	tylocalUSSMEMA.In.bUBAStat := g_tyDInput.bUBABStat;
	tylocalUSSMEMA.In.bVirtualEn := g_tyUIOut.bVSMEMAUSBEn;
	tylocalUSSMEMA.In.bUBAVirtual := g_tyUIOut.bVSMEMAUBAB;
	tylocalUSSMEMA.In.bUBAStatVirtual := g_tyUIOut.bVSMEMAUBABStat;
	tylocalUSSMEMA.In.tRstDlyTm := g_tyNtParamCurr.tUSSMEMABRstDlyTm;
	tylocalUSSMEMA.In.tSigInChkTm := g_tyNtParamCurrt.tUSSMEMAASigInChkTm;
	tylocalUSSMEMA.In.sProgNm := g_tyNtParamCurr.sUSSMEMAAProgNm;

	//Ready Receive
	IF g_tyNtParamCurr.bUSWidthChkPrep AND g_tyMcParamCurr.bUSWidthChkEn THEN
		tylocalUSSMEMA.In.bRdyRcv	:= (g_tyDInput.bnput.bUSWidthChkSen = TRUE) AND (g_tyPshrConv.bHvBrd = FALSE) AND (g_tyOpsTravLifUL.eTravLifULPosGo = TravLifULPosUS2);
	ELSE
		tylocalUSSMEMA.In.bRdyRcv	:= (g_tyPshrConv.bHvBrd = FALSE) AND (g_tyOpsTravLifUL.eTravLifULPosGo = TravLifULPosUS2) AND g_tyOps.bTravLifULUSComm;
	END_IF

	//Receive Complete Signal
	//	tylocalUSSMEMA.In.bComplSigOn	:= tylocalUSSMEMA.In.bLeftSen = FALSE;
	IF EDGENEG(tylocalUSSMEMA.In.bLeftSen) THEN
		tylocalUSSMEMA.In.bComplSigOn	:= TRUE;
	END_IF

	IF tylocalUSSMEMA.Out.eStat <> SMEMAActRun THEN
		tylocalUSSMEMA.In.bComplSigOn	:= FALSE;
	END_IF

	//Direction
	tylocalUSSMEMA.In.bDirLToR	:= g_tyNtParamCurr.eProjConvDir = ConvDirLToR OR g_tyNtParamCurr.eProjConvDir = ConvDirRToL;

	IF g_tyOps.bRun = TRUE THEN
		tylocalUSSMEMA.In.eAct := g_tyOpsTravLifUL.eUSSMEMAAct2;
	ELSIF g_tyUIOut.Out.bManualMod = TRUE THEN
		tylocalUSSMEMA.In.eAct := g_tyUIOut.eMnlAct.eUSSMEMABAct;
	ELSE
		tylocalUSSMEMA.In.eAct ACCESS ADR(eAct);
	END_IF

END_ACTION
```

#### Act_Link.st
```iecst
(** 2019-03-29 **)
ACTION Act_Link:

	//Ready Receive
	IF p_bLinkNtParamUSWidthChkPrep AND p_bLinkMcParamUSWidthChkEn THEN
		p_bRdyRcv	:= (p_bLinkDIUSWidthChkSen = TRUE) AND (p_bLinkConvHvBrd = FALSE) AND (p_eLinkOpsTravLifPosGo = TravLifULPosUS2);
	ELSE
		p_bRdyRcv	:= (p_bLinkConvHvBrd = FALSE) AND (p_eLinkOpsTravLifPosGo = TravLifULPosUS2) AND p_bLinkOpsTravLifULUSComm;
	END_IF

	//Receive Complete Signal
//	p_bComplSigOn	:= p_bLeftSen = FALSE;
	IF EDGENEG(p_bLeftSen) THEN
		p_bComplSigOn	:= TRUE;
	END_IF

	IF eStat <> SMEMAActRun THEN
		p_bComplSigOn	:= FALSE;
	END_IF

	//Direction
	p_bDirLToR	:= p_eLinkConvDir = ConvDirLToR OR p_eLinkConvDir = ConvDirLToL;

END_ACTION
```

#### Act_LinkAction.st
```iecst
(** 2019-04-09 **)
ACTION Act_LinkAction:

	IF p_bLinkOpsRun = TRUE THEN
		p_eAct ACCESS p_OpsTravLifULUSSMEMAAct2;
	ELSIF p_bManual = TRUE THEN
		p_eAct ACCESS p_UIUSSMEMABAct;
	ELSE
		p_eAct ACCESS ADR(eAct);
	END_IF

END_ACTION
```

#### Act_OutputConfig.st
```iecst
(** 2019-03-25 **)
ACTION Act_OutputConfig:

	g_tyUSSMEMAB := tylocalUSSMEMA.Out;

END_ACTION
```

#### Cyclic.st
```iecst
PROGRAM _CYCLIC

	IF bInitialDone = FALSE THEN
		IF g_tyStartUp.bNtSettingsLoadDone = TRUE THEN
			bInitialDone	:= TRUE;
			Act_Initial;
		END_IF

	ELSE

		Act_InputConfig;

		IF (tylocalUSSMEMA.In.bPrep = TRUE) AND (tylocalUSSMEMA.In.bEn = TRUE) AND (tylocalUSSMEMA.In.bDis = FALSE) THEN
			Act_Main;
		ELSE
			IF tylocalUSSMEMA.Out.eStat <> SMEMAActIdle THEN
				tylocalUSSMEMA.Out.eStatus	:= Done;
			ELSE
				tylocalUSSMEMA.Out.eStatus	:= Idle;
			END_IF
		END_IF

		Act_OutputConfig;

		Act_Alarm;

	END_IF

END_PROGRAM
```

#### Init.st
```iecst
(** 2019-03-25 **)
PROGRAM _INIT

	(* Always Change If Project Change *)

	//Pass Address To Global Address For External Use
	//Action, State & Status
	p_USSMEMABStat		:= ADR(eStat);
	p_USSMEMABStatus		:= ADR(eStatus);
	p_USSMEMABStatTxt	:= ADR(sStatTxt);

	//Alarm
	p_USSMEMABAlmData	:= ADR(tyAlmData);

	//Output
	p_USSMEMABUSRdy			:= ADR(bUSRdy);
	p_USSMEMABUSGdBrdRdy	:= ADR(bUSGdBrdRdy);
	p_USSMEMABDSRdy			:= ADR(bDSRdy);
	p_USSMEMABTransporting	:= ADR(bTransporting);
	p_USSMEMABConvStart		:= ADR(bConvStart);
	p_USSMEMABConvStop		:= ADR(bConvStop);
	p_USSMEMABUSB			:= ADR(bUSB);
	p_USSMEMABTimer			:= ADR(bTimer);
	p_USSMEMABVirtual		:= ADR(bVirtual);

	(* Always Change If Project Change *)

END_PROGRAM
```

### USSMEMA1.var - Change By Project
```iecst
VAR
	g_tyUSSMEMA1 : tyUSSMEMAAOut1;
END_VAR
(**)
```

### Program Logical/SMEMA/USSMEMA1 (IEC) - 1.00.0 - NtSMEMA v5.00.0

#### Local.var
```iecst
(*2019-04-30*)
VAR
	tylocalUSSMEMA : tyUSSMEMA;
END_VAR
(**)
(*Local Action, State & Status*)
VAR
	eAct : eSMEMAAction := SMEMAActIdle;
	eStat : eSMEMAAction := SMEMAActIdle;
	eStatus : eFBStatus := Idle;
	udiStatus : UDINT := 0;
	sStatTxt : STRING[200] := '';
	a_sStatText : ARRAY[0..50] OF STRING[200] := ['Idling','Upstream SMEMA Running','Turning On USB Signal','NA','Turning Off USB Signal','NA','Turning On USB Signal','Turning Off USB Signal',43('')];
END_VAR
(**)
(*Local Alarm*)
VAR
	tyAlmData : tyAlmDat;
	a_tyAlmText : ARRAY[10000..10099] OF tyAlmTxt := [(sAlmText:='SMEMA 9851 Transport Time Out While Transporting',sRcyText:='Timeout Expired Before Operation Completed. Reset And Resume Operation.'),(sAlmText:='SMEMA 9851 Transport Time Out After Opposite Machine Transport Finished',sRcyText:='Timeout Expired Before Operation Completed. Reset And Resume Operation.'),(sAlmText:='SMEMA 9851 Transport Time Out After Current Machine Transport Finished',sRcyText:='Timeout Expired Before Operation Completed. Reset And Resume Operation.'),(sAlmText:='SMEMA 9851 Transport Time Out After Both Machine Transport Finished And Waiting Outlet Sensor',sRcyText:='Timeout Expired Before Operation Completed. Reset And Resume Operation.'),(sAlmText:='Standard SMEMA Transport Time Out While Transporting',sRcyText:='Timeout Expired Before Operation Completed. Reset And Resume Operation.'),(sAlmText:='Standard SMEMA Transport Time Out After Opposite Machine Transport Finished',sRcyText:='Timeout Expired Before Operation Completed. Reset And Resume Operation.'),(sAlmText:='Standard SMEMA Transport Time Out After Current Machine Transport Finished',sRcyText:='Timeout Expired Before Operation Completed. Reset And Resume Operation.'),(sAlmText:='Standard SMEMA Transport Time Out After Both Machine Transport Finished And Waiting Outlet Sensor',sRcyText:='Timeout Expired Before Operation Completed. Reset And Resume Operation.'),92((0))];
END_VAR
(**)
(*Local Output*)
VAR
	bUSRdy : BOOL := FALSE;
	bUSGdBrdRdy : BOOL := FALSE;
	bDSRdy : BOOL := FALSE;
	bTransporting : BOOL := FALSE;
	bConvStart : BOOL := FALSE;
	bConvStop : BOOL := FALSE;
	bUSB : BOOL := FALSE;
	bTimer : BOOL;
	bVirtual : BOOL;
END_VAR
(**)
(*Local Input*)
VAR
	udiRstErr : UDINT := 0;
	bPrep : BOOL := TRUE;
	bEn : BOOL := TRUE;
	bDis : BOOL := FALSE;
	bManual : BOOL := FALSE;
	tyParam : tySMEMAParam;
	diTransferInTO : DINT := 20000;
	bDirLToR : BOOL := FALSE;
	bRdyRcv : BOOL := TRUE;
	bLeftSen : BOOL := FALSE;
	bRightSen : BOOL := FALSE;
	bComplSigOn : BOOL := FALSE;
	bUBA : BOOL := FALSE;
	bUBAStat : BOOL := FALSE;
	bTimerEnSen : BOOL;
	bTimerEnSenEdge : BOOL;
	bVirtualEn : BOOL;
	bUBAVirtual : BOOL;
	bUBAStatVirtual : BOOL;
	tRstDlyTm : TIME := T#500ms;
	tSigInChkTm : TIME := T#100ms;
	sProgNm : STRING[15] := 'USSMEMA';
	bNtSettingsLoadDone : BOOL := TRUE;
END_VAR
(**)
(*Local*)
VAR
	bRstErr : BOOL;
	udiRstErrOld : UDINT;
	bInitDone : BOOL;
	bInitialDone : BOOL;
	fbTimerDlyTm : TON := (PT:=T#1s);
	fbTimeTrig : R_TRIG;
	fbSMEMA_Std : fbSMEMAUS_Std;
	fbSMEMA_9851 : fbSMEMAUS_9851;
	fbSigInChk : fbSMEMASigInChk;
	eStatOld : eSMEMAAction := SMEMAActIdle;
	udiModuleNum : UDINT := 2701;
END_VAR
```

#### Act_Alarm.st
```iecst
(** 2019-03-25 **)
ACTION Act_Alarm:

	//Error
	IF EDGEPOS(eStatus = Error) THEN

		tyAlmData.sProgNm		:= p_sProgNm;
		tyAlmData.udiCode		:= udiStatus;
		tyAlmData.eSeverity		:= AlmSeverityError;
		tyAlmData.udiRunTime	:= tyAlmData.udiRunTime + 1;
		tyAlmData.bAlm			:= TRUE;
		tyAlmData.udiModuleNum  := udiModuleNum;
		g_sUSSMEMAProgNm		:= p_sProgNm;

		//Get Error Message
		IF tyAlmData.udiCode < 10000 OR tyAlmData.udiCode > 10099 THEN
			tyAlmData.sAlmMsg	:= 'Unknown';
			tyAlmData.sRcyMsg	:= 'Unknown';
		ELSE
			tyAlmData.sAlmMsg	:= a_tyAlmText[tyAlmData.udiCode].sAlmText;
			tyAlmData.sRcyMsg	:= a_tyAlmText[tyAlmData.udiCode].sRcyText;
		END_IF

		sStatTxt	:= tyAlmData.sAlmMsg;

	ELSIF bRstErr AND (tyAlmData.udiCode <> 0) THEN

		tyAlmData.udiCode	:= 0;
		tyAlmData.eSeverity	:= AlmSeverityNA;
		tyAlmData.sAlmMsg	:= '';
		tyAlmData.sRcyMsg	:= '';
		tyAlmData.bAlm			:= FALSE;
		sStatTxt	:= a_sStatText[eStat];

	END_IF

END_ACTION
```

#### Act_InitGlobal.st
```iecst
(** 2019-04-09 **)
ACTION Act_InitGlobal:

	(* Always Change If Project Change *)

	//Pass Data To Link
	p_bLinkOpsRun ACCESS p_OpsRun;
	p_bLinkNtParamProjMagConvPrep ACCESS p_NtParamProjMag1ConvPrep;

	p_eLinkConvDir ACCESS p_NtParamProjConvDir;
//	p_bLinkOpsMagMagBffrAvl ACCESS p_OpsMagUL1MagBffrAvl;
	p_bLinkOpsMagConvMagBffrAvl ACCESS p_OpsMagConvUL1MagBffrAvl;

	p_eLinkOpsLifMagULMagNxtLoad ACCESS p_OpsLifMagULMagNxtLoad;
	p_bLinkProjLifterMagPlatform ACCESS p_NtParamProjLifterMagPlatform;
	//Pass Data To Internal Use
	p_udiRstErr ACCESS p_RstErrReset;
	p_bManual ACCESS p_UIMnlMod;
	p_bLeftSen ACCESS p_DIConvRgtSen;
	p_bUBA ACCESS p_DSSMEMA1DBA;
	p_bUBAStat ACCESS p_DSSMEMA1DBAStat;
	p_tRstDlyTm ACCESS p_NtParamUSSMEMA1RstDlyTm;
	p_tSigInChkTm ACCESS p_NtParamUSSMEMA1SigInChkTm;
	p_sProgNm ACCESS p_NtParamUSSMEMA1ProgNm;
	p_bNtSettingsLoadDone ACCESS p_StartupNtSettingsLoadDone;

	(* Always Change If Project Change *)

END_ACTION
```

#### Act_InputConfig.st
```iecst
ACTION Act_InputConfig:

	(* Always Change If Project Change *)

	//Pass Data To Internal Use
	tylocalUSSMEMA.In.udiRstErr := g_tyRstErr.bReset;
	tylocalUSSMEMA.In.bLeftSen := g_tyDInput.bConvRgtSen;
	tylocalUSSMEMA.In.bUBA := g_tyDSSMEMA1.bDBA;
	tylocalUSSMEMA.In.bUBAStat := g_tyDSSMEMA1.bDBAStat;
	tylocalUSSMEMA.In.tRstDlyTm := g_tyNtParamCurr.tUSSMEMA1RstDlyTm;
	tylocalUSSMEMA.In.tSigInChkTm := g_tyNtParamCurr.tUSSMEMA1SigInChkTm;
	tylocalUSSMEMA.In.sProgNm := g_tyNtParamCurr.sUSSMEMA1ProgNm;

	(* Always Change If Project Change *)

	IF g_tyNtParamCurr.bProjLifterMagPlatform = FALSE THEN
		tylocalUSSMEMA.In.bRdyRcv	:=  g_tyOpsMagConvUL1.bMagBffrAvl = TRUE;
	ELSE
		tylocalUSSMEMA.In.bRdyRcv	:= g_tyOpsLifMagUL.eMagNxtLoad = MagNxtLoadMag1;
	END_IF

	tylocalUSSMEMA.In.bComplSigOn	:= tylocalUSSMEMA.In.bLeftSen = FALSE;

	tylocalUSSMEMA.In.bDirLToR	:= tylocalUSSMEMA.In.eLinkConvDir = ConvDirLToR OR tylocalUSSMEMA.In.eLinkConvDir = ConvDirLToL;F eStat <> SMEMAActRun THEN
		tylocalUSSMEMA.In.bComplSigOn	:= FALSE;
	END_IF

	//Direction
	tylocalUSSMEMA.In.bDirLToR	:= tylocalUSSMEMA.In.eLinkConvDir = ConvDirLToR OR tylocalUSSMEMA.In.eLinkConvDir = ConvDirLToL;

	IF tylocalUSSMEMA.In.bLinkOpsRun = TRUE THEN
		IF g_tyNtParamCurr.bProjLifterMagPlatform = FALSE THEN
			tylocalUSSMEMA.In.eAct := g_tyOpsMagConvUL1.eUSSMEMAAct;
		ELSE
			tylocalUSSMEMA.In.eAct := g_tyOpsLifMagUL.eUSSMEMAAct1;
		END_IF
	ELSE
		tylocalUSSMEMA.In.eAct := eAct;
	END_IF

END_ACTION
```

#### Act_Link.st
```iecst
(** 2019-03-29 **)
ACTION Act_Link:
	IF p_bLinkProjLifterMagPlatform = FALSE THEN
		p_bRdyRcv	:= (*p_bLinkOpsMagMagBffrAvl = TRUE OR*) p_bLinkOpsMagConvMagBffrAvl = TRUE;
	ELSE
		p_bRdyRcv	:= p_eLinkOpsLifMagULMagNxtLoad = MagNxtLoadMag1;
	END_IF

	p_bComplSigOn	:= p_bLeftSen = FALSE;

	p_bDirLToR	:= p_eLinkConvDir = ConvDirLToR OR p_eLinkConvDir = ConvDirLToL;

END_ACTION
```

#### Act_LinkAction.st
```iecst
(** 2019-04-09 **)
ACTION Act_LinkAction:

	IF p_bLinkOpsRun = TRUE THEN
		IF p_bLinkProjLifterMagPlatform = FALSE THEN
			p_eAct ACCESS p_OpsMagConvUL1USSMEMAAct;
		ELSE
			p_eAct ACCESS p_OpsLifMagULUSSMEMAAct1;
		END_IF
	ELSE
		p_eAct ACCESS ADR(eAct);
	END_IF

END_ACTION
```

#### Act_OutputConfig.st
```iecst
(** 2019-03-25 **)
ACTION Act_OutputConfig:

	g_tyUSSMEMA1 := tylocalUSSMEMA.Out;

END_ACTION
```

#### Init.st
```iecst
(** 2019-03-25 **)
PROGRAM _INIT

	(* Always Change If Project Change *)

	//Physical Configuration
	tyParam.eSelection	:= SMEMASelIPC9851;

	//Pass Address To Global Address For External Use
	//Action, State & Status
	p_USSMEMA1Stat		:= ADR(eStat);
	p_USSMEMA1Status	:= ADR(eStatus);
	p_USSMEMA1StatTxt	:= ADR(sStatTxt);

	//Alarm
	p_USSMEMA1AlmData	:= ADR(tyAlmData);

	//Output
	p_USSMEMA1USRdy			:= ADR(bUSRdy);
	p_USSMEMA1USGdBrdRdy	:= ADR(bUSGdBrdRdy);
	p_USSMEMA1DSRdy			:= ADR(bDSRdy);
	p_USSMEMA1Transporting	:= ADR(bTransporting);
	p_USSMEMA1ConvStart		:= ADR(bConvStart);
	p_USSMEMA1ConvStop		:= ADR(bConvStop);
	p_USSMEMA1USB			:= ADR(bUSB);
	p_USSMEMA1Timer			:= ADR(bTimer);
	p_USSMEMA1Virtual		:= ADR(bVirtual);

	(* Always Change If Project Change *)

END_PROGRAM
```

### USSMEMA2.var - Change By Project
```iecst
VAR
	g_tyUSSMEMA2 : tyUSSMEMAAOut1;
END_VAR
```

### Program Logical/SMEMA/USSMEMA2 (IEC) - 1.00.0 - NtSMEMA v5.00.0

#### InputRef_Link.var
```iecst
(*2019-04-09*)
(**)
(*External Data*)
VAR
	p_bLinkOpsRun : REFERENCE TO BOOL;
	p_bLinkNtParamProjMagConvPrep : REFERENCE TO BOOL;
END_VAR
(**)
VAR
	p_eLinkConvDir : REFERENCE TO eConvDir;
	p_bLinkOpsMagMagBffrAvl : REFERENCE TO BOOL;
	p_bLinkOpsMagConvMagBffrAvl : REFERENCE TO BOOL;
	p_eLinkOpsLifMagULMagNxtLoad : REFERENCE TO eLifMagULMagNxtLoad;
	p_bLinkProjLifterMagPlatform : REFERENCE TO BOOL;
END_VAR
```

#### Act_InitGlobal.st
```iecst
(** 2019-04-09 **)
ACTION Act_InitGlobal:

	(* Always Change If Project Change *)

	//Pass Data To Link
	p_bLinkOpsRun ACCESS p_OpsRun;
	p_bLinkNtParamProjMagConvPrep ACCESS p_NtParamProjMag2ConvPrep;

	p_eLinkConvDir ACCESS p_NtParamProjConvDir;
//	p_bLinkOpsMagMagBffrAvl ACCESS p_OpsMagUL2MagBffrAvl;
	p_bLinkOpsMagConvMagBffrAvl ACCESS p_OpsMagConvUL2MagBffrAvl;

	p_eLinkOpsLifMagULMagNxtLoad ACCESS p_OpsLifMagULMagNxtLoad;
	p_bLinkProjLifterMagPlatform ACCESS p_NtParamProjLifterMagPlatform;
	//Pass Data To Internal Use
	p_udiRstErr ACCESS p_RstErrReset;
	p_bManual ACCESS p_UIMnlMod;
	p_bLeftSen ACCESS p_DIConvRgtSen;
	p_bUBA ACCESS p_DSSMEMA2DBA;
	p_bUBAStat ACCESS p_DSSMEMA2DBAStat;
	p_tRstDlyTm ACCESS p_NtParamUSSMEMA2RstDlyTm;
	p_tSigInChkTm ACCESS p_NtParamUSSMEMA2SigInChkTm;
	p_sProgNm ACCESS p_NtParamUSSMEMA2ProgNm;
	p_bNtSettingsLoadDone ACCESS p_StartupNtSettingsLoadDone;

	(* Always Change If Project Change *)

END_ACTION
```

#### Act_InputConfig.st
```iecst
ACTION Act_InputConfig:

	(* Always Change If Project Change *)

	//Pass Data To Link
	tylocalUSSMEMA.In.udiRstErr := g_tyRstErr.bReset;
	tylocalUSSMEMA.In.bLeftSen := g_tyDInput.bConvRgtSen;
	tylocalUSSMEMA.In.bUBA := g_tyDSSMEMA2.bDBA;
	tylocalUSSMEMA.In.bUBAStat := g_tyDSSMEMA2.bDBAStat;
	tylocalUSSMEMA.In.tRstDlyTm := g_tyNtParamCurr.tUSSMEMA2RstDlyTm;
	tylocalUSSMEMA.In.tSigInChkTm := g_tyNtParamCurr.tUSSMEMA2SigInChkTm;
	tylocalUSSMEMA.In.sProgNm := g_tyNtParamCurr.sUSSMEMA2ProgNm;

	IF g_tyNtParamCurr.bProjLifterMagPlatform = FALSE THEN
		tylocalUSSMEMA.In.bRdyRcv	:=  g_tyOpsMagConvUL2.bMagBffrAvl = TRUE;
	ELSE
		tylocalUSSMEMA.In.bRdyRcv	:= g_tyOpsLifMagUL.eMagNxtLoad = MagNxtLoadMag2;
	END_IF

	tylocalUSSMEMA.In.bComplSigOn	:= tylocalUSSMEMA.In.bLeftSen = FALSE;

	tylocalUSSMEMA.In.bDirLToR	:= tylocalUSSMEMA.In.eLinkConvDir = ConvDirLToR OR tylocalUSSMEMA.In.eLinkConvDir = ConvDirLToL;F eStat <> SMEMAActRun THEN
	tylocalUSSMEMA.In.bComplSigOn	:= FALSE;
	END_IF

	//Direction
	tylocalUSSMEMA.In.bDirLToR	:= tylocalUSSMEMA.In.eLinkConvDir = ConvDirLToR OR tylocalUSSMEMA.In.eLinkConvDir = ConvDirLToL;

	IF tylocalUSSMEMA.In.bLinkOpsRun = TRUE THEN
		IF g_tyNtParamCurr.bProjLifterMagPlatform = FALSE THEN
			tylocalUSSMEMA.In.eAct := g_tyOpsMagConvUL2.eUSSMEMAAct;
		ELSE
			tylocalUSSMEMA.In.eAct := g_tyOpsLifMagUL.eUSSMEMAAct2;
		END_IF
	ELSE
		tylocalUSSMEMA.In.eAct := eAct;
	END_IF
END_ACTION
```

#### Act_Link.st
```iecst
(** 2019-03-29 **)
ACTION Act_Link:

	IF p_bLinkProjLifterMagPlatform = FALSE THEN
		p_bRdyRcv	:= (*p_bLinkOpsMagMagBffrAvl = TRUE OR*) p_bLinkOpsMagConvMagBffrAvl = TRUE;
	ELSE
		p_bRdyRcv	:= p_eLinkOpsLifMagULMagNxtLoad = MagNxtLoadMag2;
	END_IF

	p_bComplSigOn	:= p_bLeftSen = FALSE;

	p_bDirLToR	:= p_eLinkConvDir = ConvDirLToR OR p_eLinkConvDir = ConvDirLToL;

END_ACTION
```

#### Act_LinkAction.st
```iecst
(** 2019-04-09 **)
ACTION Act_LinkAction:

	IF p_bLinkOpsRun = TRUE THEN
		IF p_bLinkProjLifterMagPlatform = FALSE THEN
			p_eAct ACCESS p_OpsMagConvUL2USSMEMAAct;
		ELSE
			p_eAct ACCESS p_OpsLifMagULUSSMEMAAct2;
		END_IF
	ELSE
		p_eAct ACCESS ADR(eAct);
	END_IF

END_ACTION
```

#### Act_OutputConfig.st
```iecst
(** 2019-03-25 **)
ACTION Act_OutputConfig:

	g_tyUSSMEMA2 := tylocalUSSMEMA.Out;

END_ACTION
```

#### Init.st
```iecst
(** 2019-03-25 **)
PROGRAM _INIT

	(* Always Change If Project Change *)

	//Physical Configuration
	tyParam.eSelection	:= SMEMASelIPC9851;

	//Pass Address To Global Address For External Use
	//Action, State & Status
	p_USSMEMA2Stat		:= ADR(eStat);
	p_USSMEMA2Status	:= ADR(eStatus);
	p_USSMEMA2StatTxt	:= ADR(sStatTxt);

	//Alarm
	p_USSMEMA2AlmData	:= ADR(tyAlmData);

	//Output
	p_USSMEMA2USRdy			:= ADR(bUSRdy);
	p_USSMEMA2USGdBrdRdy	:= ADR(bUSGdBrdRdy);
	p_USSMEMA2DSRdy			:= ADR(bDSRdy);
	p_USSMEMA2Transporting	:= ADR(bTransporting);
	p_USSMEMA2ConvStart		:= ADR(bConvStart);
	p_USSMEMA2ConvStop		:= ADR(bConvStop);
	p_USSMEMA2USB			:= ADR(bUSB);
	p_USSMEMA2Timer			:= ADR(bTimer);
	p_USSMEMA2Virtual		:= ADR(bVirtual);

	(* Always Change If Project Change *)

END_PROGRAM
```

### USSMEMA3.var - Change By Project
```iecst
VAR
	g_tyUSSMEMA3 : tyUSSMEMAAOut1;
END_VAR
```

### Program Logical/SMEMA/USSMEMA3 (IEC) - 1.00.0 - NtSMEMA v5.00.0

#### Act_Alarm.st
```iecst
(** 2019-03-25 **)
ACTION Act_Alarm:

	//Error
	IF EDGEPOS(eStatus = Error) THEN

		tyAlmData.sProgNm		:= p_sProgNm;
		tyAlmData.udiCode		:= udiStatus;
		tyAlmData.eSeverity		:= AlmSeverityError;
		tyAlmData.udiRunTime	:= tyAlmData.udiRunTime + 1;
		tyAlmData.bAlm			:= TRUE;
		tyAlmData.udiModuleNum  := udiModuleNum;
		g_sUSSMEMAProgNm		:= p_sProgNm;

		//Get Error Message
		IF tyAlmData.udiCode < 10000 OR tyAlmData.udiCode > 10099 THEN
			tyAlmData.sAlmMsg	:= 'Unknown';
			tyAlmData.sRcyMsg	:= 'Unknown';
		ELSE
			tyAlmData.sAlmMsg	:= a_tyAlmText[tyAlmData.udiCode].sAlmText;
			tyAlmData.sRcyMsg	:= a_tyAlmText[tyAlmData.udiCode].sRcyText;
		END_IF

		sStatTxt	:= tyAlmData.sAlmMsg;

	ELSIF bRstErr AND (tyAlmData.udiCode <> 0) THEN

		tyAlmData.udiCode	:= 0;
		tyAlmData.eSeverity	:= AlmSeverityNA;
		tyAlmData.sAlmMsg	:= '';
		tyAlmData.sRcyMsg	:= '';
		tyAlmData.bAlm			:= FALSE;
		sStatTxt	:= a_sStatText[eStat];

	END_IF

END_ACTION
```

#### Act_InitGlobal.st
```iecst
(** 2019-04-09 **)
ACTION Act_InitGlobal:

	(* Always Change If Project Change *)

	//Pass Data To Link
	p_bLinkOpsRun ACCESS p_OpsRun;
	p_bLinkNtParamProjMagConvPrep ACCESS p_NtParamProjMag3ConvPrep;

	p_eLinkConvDir ACCESS p_NtParamProjConvDir;
//	p_bLinkOpsMagMagBffrAvl ACCESS p_OpsMagUL3MagBffrAvl;
	p_bLinkOpsMagConvMagBffrAvl ACCESS p_OpsMagConvUL3MagBffrAvl;

	p_eLinkOpsLifMagULMagNxtLoad ACCESS p_OpsLifMagULMagNxtLoad;
	p_bLinkProjLifterMagPlatform ACCESS p_NtParamProjLifterMagPlatform;
	//Pass Data To Internal Use
	p_udiRstErr ACCESS p_RstErrReset;
	p_bManual ACCESS p_UIMnlMod;
	p_bLeftSen ACCESS p_DIConvRgtSen;
	p_bUBA ACCESS p_DSSMEMA3DBA;
	p_bUBAStat ACCESS p_DSSMEMA3DBAStat;
	p_tRstDlyTm ACCESS p_NtParamUSSMEMA3RstDlyTm;
	p_tSigInChkTm ACCESS p_NtParamUSSMEMA3SigInChkTm;
	p_sProgNm ACCESS p_NtParamUSSMEMA3ProgNm;
	p_bNtSettingsLoadDone ACCESS p_StartupNtSettingsLoadDone;

	(* Always Change If Project Change *)

END_ACTION
```

#### Act_InputConfig.st
```iecst
ACTION Act_InputConfig:

	(* Always Change If Project Change *)

	//Pass Data To Link
	tylocalUSSMEMA.In.udiRstErr := g_tyRstErr.bReset;
	tylocalUSSMEMA.In.bLeftSen := g_tyDInput.bConvRgtSen;
	tylocalUSSMEMA.In.bUBA := g_tyDSSMEMA3.bDBA;
	tylocalUSSMEMA.In.bUBAStat := g_tyDSSMEMA3.bDBAStat;
	tylocalUSSMEMA.In.tRstDlyTm := g_tyNtParamCurr.tUSSMEMA3RstDlyTm;
	tylocalUSSMEMA.In.tSigInChkTm := g_tyNtParamCurr.tUSSMEMA3SigInChkTm;
	tylocalUSSMEMA.In.sProgNm := g_tyNtParamCurr.sUSSMEMA3ProgNm;

	IF g_tyNtParamCurr.bProjLifterMagPlatform = FALSE THEN
		tylocalUSSMEMA.In.bRdyRcv	:=  g_tyOpsMagConvUL3.bMagBffrAvl = TRUE;
	ELSE
		tylocalUSSMEMA.In.bRdyRcv	:= g_tyOpsLifMagUL.eMagNxtLoad = MagNxtLoadMag3;
	END_IF

	tylocalUSSMEMA.In.bComplSigOn	:= tylocalUSSMEMA.In.bLeftSen = FALSE;

	tylocalUSSMEMA.In.bDirLToR	:= tylocalUSSMEMA.In.eLinkConvDir = ConvDirLToR OR tylocalUSSMEMA.In.eLinkConvDir = ConvDirLToL;F eStat <> SMEMAActRun THEN
	tylocalUSSMEMA.In.bComplSigOn	:= FALSE;
	END_IF

	//Direction
	tylocalUSSMEMA.In.bDirLToR	:= tylocalUSSMEMA.In.eLinkConvDir = ConvDirLToR OR tylocalUSSMEMA.In.eLinkConvDir = ConvDirLToL;

	IF tylocalUSSMEMA.In.bLinkOpsRun = TRUE THEN
		IF g_tyNtParamCurr.bProjLifterMagPlatform = FALSE THEN
			tylocalUSSMEMA.In.eAct := g_tyOpsMagConvUL3.eUSSMEMAAct;
		ELSE
			tylocalUSSMEMA.In.eAct := g_tyOpsLifMagUL.eUSSMEMAAct3;
		END_IF
	ELSE
		tylocalUSSMEMA.In.eAct := eAct;
	END_IF

END_ACTION
```

#### Act_Link.st
```iecst
(** 2019-03-29 **)
ACTION Act_Link:

	IF p_bLinkProjLifterMagPlatform = FALSE THEN
		p_bRdyRcv	:= (*p_bLinkOpsMagMagBffrAvl = TRUE OR*) p_bLinkOpsMagConvMagBffrAvl = TRUE;
	ELSE
		p_bRdyRcv	:= p_eLinkOpsLifMagULMagNxtLoad = MagNxtLoadMag3;
	END_IF

	p_bComplSigOn	:= p_bLeftSen = FALSE;

	p_bDirLToR	:= p_eLinkConvDir = ConvDirLToR OR p_eLinkConvDir = ConvDirLToL;

END_ACTION
```

#### Act_LinkAction.st
```iecst
(** 2019-04-09 **)
ACTION Act_LinkAction:

	IF p_bLinkOpsRun = TRUE THEN
		IF p_bLinkProjLifterMagPlatform = FALSE THEN
			p_eAct ACCESS p_OpsMagConvUL3USSMEMAAct;
		ELSE
			p_eAct ACCESS p_OpsLifMagULUSSMEMAAct3;
		END_IF
	ELSE
		p_eAct ACCESS ADR(eAct);
	END_IF

END_ACTION
```

#### Act_OutputConfig.st
```iecst
(** 2019-03-25 **)
ACTION Act_OutputConfig:

	g_tyUSSMEMA3 := tylocalUSSMEMA.Out;

END_ACTION
```

#### Init.st
```iecst
(** 2019-03-25 **)
PROGRAM _INIT

	(* Always Change If Project Change *)

	//Physical Configuration
	tyParam.eSelection	:= SMEMASelIPC9851;

	//Pass Address To Global Address For External Use
	//Action, State & Status
	p_USSMEMA3Stat		:= ADR(eStat);
	p_USSMEMA3Status	:= ADR(eStatus);
	p_USSMEMA3StatTxt	:= ADR(sStatTxt);

	//Alarm
	p_USSMEMA3AlmData	:= ADR(tyAlmData);

	//Output
	p_USSMEMA3USRdy			:= ADR(bUSRdy);
	p_USSMEMA3USGdBrdRdy	:= ADR(bUSGdBrdRdy);
	p_USSMEMA3DSRdy			:= ADR(bDSRdy);
	p_USSMEMA3Transporting	:= ADR(bTransporting);
	p_USSMEMA3ConvStart		:= ADR(bConvStart);
	p_USSMEMA3ConvStop		:= ADR(bConvStop);
	p_USSMEMA3USB			:= ADR(bUSB);
	p_USSMEMA3Timer			:= ADR(bTimer);
	p_USSMEMA3Virtual		:= ADR(bVirtual);

	(* Always Change If Project Change *)

END_PROGRAM
```

### DSSMEMA1.var - Change By Project
```iecst
(*2019-03-25*)
VAR
	g_tyDSSMEMA1 : tyDSSMEMAOut1;
END_VAR
```

### Program Logical/SMEMA/DSSMEMA1 (IEC) - 1.00.0 - NtSMEMA v5.00.0

#### Act_Background.st
```iecst
(** 2019-01-20 **)
ACTION Act_Background:

	fbTimeTrig(CLK := p_bTimerEnSenEdge);

	IF eStat = SMEMAActRun AND (p_bTimerEnSenEdge OR p_bTimerEnSen) THEN
		IF fbTimeTrig.Q = TRUE OR p_bTimerEnSen THEN
			fbTimerDlyTm.IN	:= TRUE;
		END_IF
	ELSE
		fbTimerDlyTm.IN	:= FALSE;
	END_IF

	IF bConvStart = FALSE AND bConvStop = FALSE THEN
		fbTimerDlyTm;

		IF fbTimerDlyTm.Q = TRUE AND eStat = SMEMAActRun THEN
			bTimer		:= TRUE;
			bVirtual	:= FALSE;
		ELSIF p_bVirtualEn = TRUE THEN
			bTimer		:= FALSE;
			bVirtual	:= TRUE;
		ELSE
			bTimer		:= FALSE;
			bVirtual	:= FALSE;
		END_IF
	ELSE
		fbTimerDlyTm(IN := FALSE);
	END_IF

	IF bTimer = TRUE THEN

		fbSigInChk.bNomSig			:= bConvStart = FALSE AND bConvStop = FALSE;
		fbSigInChk.bStatSig			:= FALSE;
		fbSigInChk.bStatSigSetGd	:= FALSE;

	ELSIF bVirtual = TRUE THEN

		fbSigInChk.bNomSig			:= p_bDSBVirtual;
		fbSigInChk.bStatSig			:= FALSE;
		fbSigInChk.bStatSigSetGd	:= FALSE;

	ELSE

		fbSigInChk.bNomSig			:= p_bDSB;
		fbSigInChk.bStatSig			:= FALSE;
		fbSigInChk.bStatSigSetGd	:= FALSE;

	END_IF

	fbSigInChk;

	bDSRdy	:= fbSigInChk.bSigInValid;
//	bDSTransportFinished := bConvStart AND EDGENEG(p_bRightSen); //bDBA = FALSE
END_ACTION
```

#### Act_InitGlobal.st
```iecst
(** 2019-04-09 **)
ACTION Act_InitGlobal:

	(* Always Change If Project Change *)

	//Pass Data To Link
	p_bLinkOpsRun ACCESS p_OpsRun;

	p_bLinkConvHvBrd ACCESS p_PshrConvHvBrd;
	p_eLinkConvDir ACCESS p_NtParamProjConvDir;
	p_eLinkOpsTravLifPosGo ACCESS p_OpsTravLifULPosGo;

	//Pass Data To Internal Use
	p_udiRstErr ACCESS p_RstErrReset;
	p_bManual ACCESS p_UIMnlMod;
	p_bGdBrd ACCESS p_PshrConvGdBrd;
	p_bLeftSen ACCESS p_DIConvLftSen;
	p_bRightSen ACCESS p_DIConvRgtSen;
	p_bClrSen ACCESS p_DIConvClrSen;
	p_bDSB ACCESS p_USSMEMA1USB;
	p_tRstDlyTm ACCESS p_NtParamDSSMEMA1RstDlyTm;
	p_tSigInChkTm ACCESS p_NtParamDSSMEMA1SigInChkTm;
	p_sProgNm ACCESS p_NtParamDSSMEMA1ProgNm;
	p_bNtSettingsLoadDone ACCESS p_StartupNtSettingsLoadDone;

	(* Always Change If Project Change *)

END_ACTION
```

#### Act_Initial.st
```iecst
(** 2019-04-27 **)
ACTION Act_Initial:

	//Initial
	tylocalDSSMEMA.Out.sStatTxt	:= a_sStatText[eStat];

	fbSMEMA_OppFirst.tRstDlyTm	:= tylocalDSSMEMA.In.tRstDlyTm;
	fbSMEMA_OppFirst(bEn := FALSE);

	fbSMEMA.tRstDlyTm	:= tylocalDSSMEMA.In.tRstDlyTm;
	fbSMEMA(bEn := FALSE);

	fbTimerDlyTm(IN := FALSE);
	fbTimeTrig(CLK := TRUE);

	fbSigInChk.tSigInChkTm	:= tylocalDSSMEMA.In.tSigInChkTm;

END_ACTION
```

#### Act_InputConfig.st
```iecst
(** 2019-04-09 **)
ACTION Act_InputConfig:

	(* Always Change If Project Change *)

	//Pass Data To Link
	tylocalDSSMEMA.In.udiRstErr := g_tyRstErrOut.udiRstErr;
	tylocalDSSMEMA.In.bGdBrd := g_tyPshrConvGdBrd;
	tylocalDSSMEMA.In.bLeftSen := g_tyDInput.bConvLftSen;
	tylocalDSSMEMA.In.bRightSen := g_tyDInput.bConvRgtSen;
	tylocalDSSMEMA.In.bClrSen := g_tyDInput.bConvClrSen;
	tylocalDSSMEMA.In.bDSB := g_tyUSSMEMA1.bUSB;
	tylocalDSSMEMA.In.tRstDlyTm := g_tyNtParamCurr.tDSSMEMA1RstDlyTm;
	tylocalDSSMEMA.In.tSigInChkTm := g_tyNtParamCurr.tDSSMEMA1SigInChkTm;
	tylocalDSSMEMA.In.sProgNm := g_tyNtParamCurr.sDSSMEMA1ProgNm;

	(tylocalDSSMEMA.In.bRdySend	:= g_tyPshrConv.bHvBrd AND g_tyOpsTravLifUL.eTravLifULPosGo = TravLifULPosDS1;

	tylocalDSSMEMA.In.bComplSigOn	:= g_tyPshrConv.bHvBrd = FALSE AND tylocalDSSMEMA.In.bClrSen = FALSE;

	tylocalDSSMEMA.In.bDirLToR	:= g_tyNtParamCurr.eProjConvDir = ConvDirLToR OR g_tyNtParamCurr.eProjConvDir = ConvDirLToL;

	IF g_tyOps.bRun = TRUE THEN
		tylocalDSSMEMA.In.eAct := g_tyOpsTravLifULDSSMEMAAct1;
	ELSE
		tylocalDSSMEMA.In.eAct ACCESS ADR(eAct);
	END_IF

END_ACTION
```

#### Act_Link.st
```iecst
(** 2019-03-29 **)
ACTION Act_Link:

	p_bRdySend	:= p_bLinkConvHvBrd AND p_eLinkOpsTravLifPosGo = TravLifULPosDS1;

	p_bComplSigOn	:= p_bLinkConvHvBrd = FALSE AND p_bClrSen = FALSE;

	p_bDirLToR	:= p_eLinkConvDir = ConvDirLToR OR p_eLinkConvDir = ConvDirLToL;

END_ACTION
```

#### Act_LinkAction.st
```iecst
(** 2019-04-09 **)
ACTION Act_LinkAction:

	IF p_bLinkOpsRun = TRUE THEN
		p_eAct ACCESS p_OpsTravLifULDSSMEMAAct1;
	ELSE
		p_eAct ACCESS ADR(eAct);
	END_IF

END_ACTION
```

#### Act_OutputConfig.st
```iecst
(** 2019-03-25 **)
ACTION Act_OutputConfig:

	(* Always Change If Project Change *)
	g_tyDSSMEMA1 := tylocalDSSMEMA.Out;

	(* Always Change If Project Change *)

END_ACTION
```

#### Init.st
```iecst
(** 2019-03-25 **)
PROGRAM _INIT

	(* Always Change If Project Change *)

	//Physical Configuration
	tyParam.eSelection	:= SMEMASelIPC9851;

	//Pass Address To Global Address For External Use
	//Action, State & Status
	p_DSSMEMA1Stat		:= ADR(eStat);
	p_DSSMEMA1Status	:= ADR(eStatus);
	p_DSSMEMA1StatTxt	:= ADR(sStatTxt);

	//Alarm
	p_DSSMEMA1AlmData	:= ADR(tyAlmData);

	//Output
	p_DSSMEMA1USRdy			:= ADR(bUSRdy);
	p_DSSMEMA1USGdBrdRdy	:= ADR(bUSGdBrdRdy);
	p_DSSMEMA1DSRdy			:= ADR(bDSRdy);
	p_DSSMEMA1Transporting	:= ADR(bTransporting);
	p_DSSMEMA1ConvStart		:= ADR(bConvStart);
	p_DSSMEMA1ConvStop		:= ADR(bConvStop);
	p_DSSMEMA1DBA			:= ADR(bDBA);
	p_DSSMEMA1DBAStat		:= ADR(bDBAStat);
	p_DSSMEMA1Timer			:= ADR(bTimer);
	p_DSSMEMA1Virtual		:= ADR(bVirtual);

	//Svy Hermes
//	p_DSSMEMA1TransprtFinished	:= ADR(bDSTransportFinished);

	(* Always Change If Project Change *)

END_PROGRAM
```

### DSSMEMA2.var - Change By Project
```iecst
(*2019-03-25*)
VAR
	g_tyDSSMEMA2 : tyDSSMEMAOut1;
END_VAR
```

### Program Logical/SMEMA/DSSMEMA2 (IEC) - 1.00.0 - NtSMEMA v5.00.0

#### InputRef.var
```iecst
(*2019-03-25*)
(**)
(*General*)
VAR
	p_eAct : REFERENCE TO eSMEMAAction;
	p_udiRstErr : REFERENCE TO UDINT;
	p_bPrep : REFERENCE TO BOOL;
	p_bEn : REFERENCE TO BOOL;
	p_bDis : REFERENCE TO BOOL;
END_VAR
(**)
(*Configuration*)
VAR
	p_bManual : REFERENCE TO BOOL;
	p_tyParam : REFERENCE TO tySMEMAParam;
	p_bGdBrd : REFERENCE TO BOOL;
	p_diTransferOutTO : REFERENCE TO DINT;
	p_bDirLToR : REFERENCE TO BOOL;
	p_bRdySend : REFERENCE TO BOOL;
END_VAR
(**)
(*Input*)
VAR
	p_bLeftSen : REFERENCE TO BOOL;
	p_bRightSen : REFERENCE TO BOOL;
	p_bClrSen : REFERENCE TO BOOL;
	p_bComplSigOn : REFERENCE TO BOOL;
	p_bDSB : REFERENCE TO BOOL;
	p_bTimerEnSen : REFERENCE TO BOOL;
	p_bTimerEnSenEdge : REFERENCE TO BOOL;
	p_bVirtualEn : REFERENCE TO BOOL;
	p_bDSBVirtual : REFERENCE TO BOOL;
	p_tRstDlyTm : REFERENCE TO TIME;
	p_tSigInChkTm : REFERENCE TO TIME;
	p_sProgNm : REFERENCE TO STRING[15];
	p_bNtSettingsLoadDone : REFERENCE TO BOOL;
END_VAR
```

#### Local.var
```iecst
(*2019-04-30*)
VAR
	tylocalDSSMEMA : tyDSSMEMA;
END_VAR
(**)
(*Local Action, State & Status*)
VAR
	udiStatus : UDINT := 0;
	a_sStatText : ARRAY[0..50] OF STRING[200] := ['Idling','SMEMA Running','Turning On DBA Signal','Turning On DBA Stat Signal','Turning Off DBA Signal','Turning Off DBA Stat Signal','Turning On All DBA Signal','Turning Off All DBA Signal',43('')];
END_VAR
(**)
(**)
(**)
(*Local*)
VAR
	bRstErr : BOOL;
	udiRstErrOld : UDINT;
	bInitDone : BOOL;
	bInitialDone : BOOL;
	fbTimerDlyTm : TON := (PT:=T#1s);
	fbTimeTrig : R_TRIG;
	fbSMEMA_OppFirst : fbSMEMADS_OppFirst;
	fbSMEMA : fbSMEMADS;
	fbSigInChk : fbSMEMASigInChk;
	eStatOld : eSMEMAAction := SMEMAActIdle;
	udiModuleNum : UDINT := 2801;
END_VAR
```

#### Act_Alarm.st
```iecst
(** 2019-03-25 **)
ACTION Act_Alarm:

	IF tylocalDSSMEMA.In.udiRstErr <> udiRstErrOld THEN
		bRstErr			:= TRUE;
		udiRstErrOld	:= tylocalDSSMEMA.In.udiRstErr;
	ELSE
		bRstErr			:= FALSE;
	END_IF

	//Reset Error
	IF (tylocalDSSMEMA.Out.eStatus = Error) AND bRstErr THEN
		tylocalDSSMEMA.In.eAct	:= SMEMAActIdle;
		tylocalDSSMEMA.Out.eStat:= SMEMAActIdle;
	END_IF

	//Error
	IF EDGEPOS(tylocalDSSMEMA.Out.eStatus = Error) THEN

		tylocalDSSMEMA.Out.tyAlmData.sProgNm		:= tylocalDSSMEMA.In.sProgNm;
		tylocalDSSMEMA.Out.tyAlmData.udiCode		:= udiStatus;
		tylocalDSSMEMA.Out.tyAlmData.eSeverity		:= AlmSeverityError;
		tylocalDSSMEMA.Out.tyAlmData.udiRunTime		:= tylocalDSSMEMA.Out.tyAlmData.udiRunTime + 1;
		tylocalDSSMEMA.Out.tyAlmData.bAlm			:= TRUE;
		tylocalDSSMEMA.Out.tyAlmData.udiModuleNum  := udiModuleNum;
		g_sDSSMEMAProgNm		:= tylocalDSSMEMA.In.sProgNm;

	ELSIF bRstErr AND (tylocalDSSMEMA.Out.tyAlmData.udiCode <> 0) THEN

		tylocalDSSMEMA.Out.tyAlmData.udiCode	:= 0;
		tylocalDSSMEMA.Out.tyAlmData.eSeverity	:= AlmSeverityNA;
		tylocalDSSMEMA.Out.tyAlmData.bAlm		:= FALSE;

		tylocalDSSMEMA.Out.sStatTxt	:= a_sStatText[tylocalDSSMEMA.Out.eStat];

	END_IF

END_ACTION
```

#### Act_Background.st
```iecst
(** 2019-01-20 **)
ACTION Act_Background:

	fbTimeTrig(CLK := p_bTimerEnSenEdge);

	IF eStat = SMEMAActRun AND (p_bTimerEnSenEdge OR p_bTimerEnSen) THEN
		IF fbTimeTrig.Q = TRUE OR p_bTimerEnSen THEN
			fbTimerDlyTm.IN	:= TRUE;
		END_IF
	ELSE
		fbTimerDlyTm.IN	:= FALSE;
	END_IF

	IF bConvStart = FALSE AND bConvStop = FALSE THEN
		fbTimerDlyTm;

		IF fbTimerDlyTm.Q = TRUE AND eStat = SMEMAActRun THEN
			bTimer		:= TRUE;
			bVirtual	:= FALSE;
		ELSIF p_bVirtualEn = TRUE THEN
			bTimer		:= FALSE;
			bVirtual	:= TRUE;
		ELSE
			bTimer		:= FALSE;
			bVirtual	:= FALSE;
		END_IF
	ELSE
		fbTimerDlyTm(IN := FALSE);
	END_IF

	IF bTimer = TRUE THEN

		fbSigInChk.bNomSig			:= bConvStart = FALSE AND bConvStop = FALSE;
		fbSigInChk.bStatSig			:= FALSE;
		fbSigInChk.bStatSigSetGd	:= FALSE;

	ELSIF bVirtual = TRUE THEN

		fbSigInChk.bNomSig			:= p_bDSBVirtual;
		fbSigInChk.bStatSig			:= FALSE;
		fbSigInChk.bStatSigSetGd	:= FALSE;

	ELSE

		fbSigInChk.bNomSig			:= p_bDSB;
		fbSigInChk.bStatSig			:= FALSE;
		fbSigInChk.bStatSigSetGd	:= FALSE;

	END_IF

	fbSigInChk;

	bDSRdy	:= fbSigInChk.bSigInValid;
//	bDSTransportFinished := bConvStart AND EDGENEG(p_bRightSen);

END_ACTION
```

#### Act_InitGlobal.st
```iecst
(** 2019-04-09 **)
ACTION Act_InitGlobal:

	(* Always Change If Project Change *)

	//Pass Data To Link
	p_bLinkOpsRun ACCESS p_OpsRun;

	p_bLinkConvHvBrd ACCESS p_PshrConvHvBrd;
	p_eLinkConvDir ACCESS p_NtParamProjConvDir;
	p_eLinkOpsTravLifPosGo ACCESS p_OpsTravLifULPosGo;

	//Pass Data To Internal Use
	p_udiRstErr ACCESS p_RstErrReset;
	p_bManual ACCESS p_UIMnlMod;
	p_bGdBrd ACCESS p_PshrConvGdBrd;
	p_bLeftSen ACCESS p_DIConvLftSen;
	p_bRightSen ACCESS p_DIConvRgtSen;
	p_bClrSen ACCESS p_DIConvClrSen;
	p_bDSB ACCESS p_USSMEMA2USB;
	p_tRstDlyTm ACCESS p_NtParamDSSMEMA2RstDlyTm;
	p_tSigInChkTm ACCESS p_NtParamDSSMEMA2SigInChkTm;
	p_sProgNm ACCESS p_NtParamDSSMEMA2ProgNm;
	p_bNtSettingsLoadDone ACCESS p_StartupNtSettingsLoadDone;

	(* Always Change If Project Change *)

END_ACTION
```

#### Act_InputConfig.st
```iecst
(** 2019-04-09 **)
ACTION Act_InputConfig:

	(* Always Change If Project Change *)

	//Pass Data To Link
	tylocalDSSMEMA.In.udiRstErr := g_tyRstErrOut.udiRstErr;
	tylocalDSSMEMA.In.bGdBrd := g_tyPshrConvGdBrd;
	tylocalDSSMEMA.In.bLeftSen := g_tyDInput.bConvLftSen;
	tylocalDSSMEMA.In.bRightSen := g_tyDInput.bConvRgtSen;
	tylocalDSSMEMA.In.bClrSen := g_tyDInput.bConvClrSen;
	tylocalDSSMEMA.In.bDSB := g_tyUSSMEMA2.bUSB;
	tylocalDSSMEMA.In.tRstDlyTm := g_tyNtParamCurr.tDSSMEMA2RstDlyTm;
	tylocalDSSMEMA.In.tSigInChkTm := g_tyNtParamCurr.tDSSMEMA2SigInChkTm;
	tylocalDSSMEMA.In.sProgNm := g_tyNtParamCurr.sDSSMEMA2ProgNm;

	(tylocalDSSMEMA.In.bRdySend	:= g_tyPshrConv.bHvBrd AND g_tyOpsTravLifUL.eTravLifULPosGo = TravLifULPosDS2;

	tylocalDSSMEMA.In.bComplSigOn	:= g_tyPshrConv.bHvBrd = FALSE AND tylocalDSSMEMA.In.bClrSen = FALSE;

	tylocalDSSMEMA.In.bDirLToR	:= g_tyNtParamCurr.eProjConvDir = ConvDirLToR OR g_tyNtParamCurr.eProjConvDir = ConvDirLToL;

	IF g_tyOps.bRun = TRUE THEN
		tylocalDSSMEMA.In.eAct := g_tyOpsTravLifULDSSMEMAAct2;
	ELSE
		tylocalDSSMEMA.In.eAct ACCESS ADR(eAct);
	END_IF

	(* Always Change If Project Change *)

END_ACTION
```

#### Act_Link.st
```iecst
(** 2019-03-29 **)
ACTION Act_Link:

	p_bRdySend	:= p_bLinkConvHvBrd AND p_eLinkOpsTravLifPosGo = TravLifULPosDS2;

	p_bComplSigOn	:= p_bLinkConvHvBrd = FALSE AND p_bClrSen = FALSE;

	p_bDirLToR	:= p_eLinkConvDir = ConvDirLToR OR p_eLinkConvDir = ConvDirLToL;

END_ACTION
```

#### Act_LinkAction.st
```iecst
(** 2019-04-09 **)
ACTION Act_LinkAction:

	IF p_bLinkOpsRun = TRUE THEN
		p_eAct ACCESS p_OpsTravLifULDSSMEMAAct2;
	ELSE
		p_eAct ACCESS ADR(eAct);
	END_IF

END_ACTION
```

#### Act_Main.st
```iecst
ACTION Act_Main:

	fbSMEMA_OppFirst.tRstDlyTm	:= tylocalDSSMEMA.In.tRstDlyTm;
	fbSMEMA.tRstDlyTm			:= tylocalDSSMEMA.In.tRstDlyTm;
	fbSigInChk.tSigInChkTm		:= tylocalDSSMEMA.In.tSigInChkTm;

	//Timer Running
	fbTimeTrig(CLK := tylocalDSSMEMA.In.bTimerEnSenEdge);

	IF tylocalDSSMEMA.Out.eStat = SMEMAActRun AND (tylocalDSSMEMA.In.bTimerEnSenEdge OR tylocalDSSMEMA.In.bTimerEnSen) THEN
		IF fbTimeTrig.Q = TRUE OR tylocalDSSMEMA.In.bTimerEnSen THEN
			fbTimerDlyTm.IN	:= TRUE;
		END_IF
	ELSE
		fbTimerDlyTm.IN	:= FALSE;
	END_IF

	IF tylocalDSSMEMA.Out.bConvStart = FALSE AND tylocalDSSMEMA.Out.bConvStop = FALSE THEN
		fbTimerDlyTm;

		IF fbTimerDlyTm.Q = TRUE AND tylocalDSSMEMA.Out.eStat = SMEMAActRun THEN
			tylocalDSSMEMA.Out.bTimer		:= TRUE;
			tylocalDSSMEMA.Out.bVirtual	:= FALSE;
		ELSIF tylocalDSSMEMA.In.bVirtualEn = TRUE THEN
			tylocalDSSMEMA.Out.bTimer		:= FALSE;
			tylocalDSSMEMA.Out.bVirtual	:= TRUE;
		ELSE
			tylocalDSSMEMA.Out.bTimer		:= FALSE;
			tylocalDSSMEMA.Out.bVirtual	:= FALSE;
		END_IF
	ELSE
		fbTimerDlyTm(IN := FALSE);
	END_IF

	IF tylocalDSSMEMA.Out.bTimer = TRUE THEN

		fbSigInChk.bNomSig			:= tylocalDSSMEMA.Out.bConvStart = FALSE AND tylocalDSSMEMA.Out.bConvStop = FALSE;
		fbSigInChk.bStatSig			:= FALSE;
		fbSigInChk.bStatSigSetGd	:= FALSE;

	ELSIF tylocalDSSMEMA.Out.bVirtual = TRUE THEN

		fbSigInChk.bNomSig			:= tylocalDSSMEMA.In.bDSBVirtual;
		fbSigInChk.bStatSig			:= FALSE;
		fbSigInChk.bStatSigSetGd	:= FALSE;

	ELSE

		fbSigInChk.bNomSig			:= tylocalDSSMEMA.In.bDSB;
		fbSigInChk.bStatSig			:= FALSE;
		fbSigInChk.bStatSigSetGd	:= FALSE;

	END_IF

	fbSigInChk;

	tylocalDSSMEMA.Out.bDSRdy	:= fbSigInChk.bSigInValid;

	//Set tylocalDSSMEMA.In.eAct
	IF tylocalDSSMEMA.Out.eStatus = Idle OR tylocalDSSMEMA.Out.eStatus = Busy OR tylocalDSSMEMA.Out.eStatus = Done THEN
		tylocalDSSMEMA.Out.eStat	:= tylocalDSSMEMA.In.eAct;
	END_IF
	//Transition State
	IF eStatOld <> tylocalDSSMEMA.Out.eStat THEN
		fbSMEMA_OppFirst(bEn := FALSE);
		fbSMEMA(bEn := FALSE);

		tylocalDSSMEMA.Out.bTransporting	:= FALSE;
		tylocalDSSMEMA.Out.bConvStart		:= FALSE;
		tylocalDSSMEMA.Out.bConvStop		:= FALSE;
		tylocalDSSMEMA.Out.bUSRdy			:= FALSE;
		tylocalDSSMEMA.Out.bUSGdBrdRdy		:= FALSE;

		IF eStatOld <> SMEMAActIdle
			AND eStatOld <> SMEMAActSetSig
			AND eStatOld <> SMEMAActSetStatSig
			AND eStatOld <> SMEMAActRstSig
			AND eStatOld <> SMEMAActRstStatSig
			AND eStatOld <> SMEMAActSetAllSig
			AND eStatOld <> SMEMAActRstAllSig THEN

			tylocalDSSMEMA.Out.bDBA		:= FALSE;
			tylocalDSSMEMA.Out.bDBAStat	:= FALSE;

		END_IF

		tylocalDSSMEMA.Out.sStatTxt	:= a_sStatText[tylocalDSSMEMA.Out.eStat];

		eStatOld	:= tylocalDSSMEMA.Out.eStat;

		tylocalDSSMEMA.Out.eStatus		:= Busy;
	END_IF

	//Main
	CASE tylocalDSSMEMA.Out.eStat OF

		SMEMAActIdle:
			IF EDGENEG(tylocalDSSMEMA.In.bManual) THEN
				tylocalDSSMEMA.Out.bDBA		:= FALSE;
				tylocalDSSMEMA.Out.bDBAStat	:= FALSE;
			END_IF

			tylocalDSSMEMA.Out.eStatus	:= Idle;

		SMEMAActRun:
			IF tylocalDSSMEMA.Out.eStatus = Idle OR tylocalDSSMEMA.Out.eStatus = Busy THEN

				tylocalDSSMEMA.Out.eStatus	:= Busy;

				IF tylocalDSSMEMA.In.tyParam.eSelection <> SMEMASelStandard THEN

					fbSMEMA.bDSRdy		:= fbSigInChk.bSigInValid;
					fbSMEMA.bRdySend	:= tylocalDSSMEMA.In.bRdySend;
					fbSMEMA.bComplSigOn	:= tylocalDSSMEMA.In.bComplSigOn;

					fbSMEMA.tTimeOut	:= DINT_TO_TIME(tylocalDSSMEMA.In.diTransferOutTO);
					fbSMEMA(bEn := TRUE);

					tylocalDSSMEMA.Out.bTransporting	:= fbSMEMA.tylocalDSSMEMA.Out.bTransporting;
					tylocalDSSMEMA.Out.bConvStart		:= fbSMEMA.tylocalDSSMEMA.Out.bConvStart;
					tylocalDSSMEMA.Out.bConvStop		:= fbSMEMA.tylocalDSSMEMA.Out.bConvStop;
					tylocalDSSMEMA.Out.bDBA			:= fbSMEMA.bSigToDS AND (tylocalDSSMEMA.Out.bTimer = FALSE) AND (tylocalDSSMEMA.Out.bVirtual = FALSE);
					tylocalDSSMEMA.Out.bDBAStat		:= (fbSMEMA.bSigToDS) AND (fSMEMASigStatOut(tylocalDSSMEMA.In.tyParam.bStatSigSetGd, tylocalDSSMEMA.In.bGdBrd)) AND (tylocalDSSMEMA.In.tyParam.eSelection = SMEMASelIPC9851Ext);

					tylocalDSSMEMA.Out.bUSRdy			:= fbSMEMA.bSigToDS;
					tylocalDSSMEMA.Out.bUSGdBrdRdy		:= tylocalDSSMEMA.In.bGdBrd;

					IF fbSMEMA.udiStatus = 0 THEN
						tylocalDSSMEMA.Out.eStatus	:= Done;
					ELSIF fbSMEMA.udiStatus < 65534 THEN
						tylocalDSSMEMA.Out.eStatus		:= Error;

						IF fbSMEMA.udiStatus = 1200 THEN
							udiStatus	:= 10000;	//SMEMA 9851 Transport Time Out While Transporting
						ELSIF fbSMEMA.udiStatus = 1201 THEN
							udiStatus	:= 10001;	//SMEMA 9851 Transport Time Out After Opposite Machine Transport Finished
						ELSIF fbSMEMA.udiStatus = 1202 THEN
							udiStatus	:= 10002;	//SMEMA 9851 Transport Time Out After Current Machine Transport Finished
						ELSIF fbSMEMA.udiStatus = 1203 THEN
							udiStatus	:= 10003;	//SMEMA 9851 Transport Time Out After Both Machine Transport Finished And Waiting Outlet Sensor
						ELSE
							udiStatus	:= fbSMEMA.udiStatus;
						END_IF
					END_IF

				ELSE

					fbSMEMA_OppFirst.bDSRdy			:= fbSigInChk.bSigInValid;
					fbSMEMA_OppFirst.bRdySend		:= tylocalDSSMEMA.In.bRdySend;
					fbSMEMA_OppFirst.bComplSigOn	:= tylocalDSSMEMA.In.bComplSigOn;

					fbSMEMA_OppFirst.tTimeOut	:= DINT_TO_TIME(tylocalDSSMEMA.In.diTransferOutTO);
					fbSMEMA_OppFirst(bEn := TRUE);

					tylocalDSSMEMA.Out.bTransporting	:= fbSMEMA_OppFirst.tylocalDSSMEMA.Out.bTransporting;
					tylocalDSSMEMA.Out.bConvStart		:= fbSMEMA_OppFirst.tylocalDSSMEMA.Out.bConvStart;
					tylocalDSSMEMA.Out.bConvStop		:= fbSMEMA_OppFirst.tylocalDSSMEMA.Out.bConvStop;
					tylocalDSSMEMA.Out.bDBA			:= fbSMEMA_OppFirst.bSigToDS AND (tylocalDSSMEMA.Out.bTimer = FALSE) AND (tylocalDSSMEMA.Out.bVirtual = FALSE);
					tylocalDSSMEMA.Out.bDBAStat		:= (fbSMEMA_OppFirst.bSigToDS) AND (fSMEMASigStatOut(tylocalDSSMEMA.In.tyParam.bStatSigSetGd, tylocalDSSMEMA.In.bGdBrd)) AND (tylocalDSSMEMA.In.tyParam.eSelection = SMEMASelIPC9851Ext);

					tylocalDSSMEMA.Out.bUSRdy			:= fbSMEMA_OppFirst.bSigToDS;
					tylocalDSSMEMA.Out.bUSGdBrdRdy		:= tylocalDSSMEMA.In.bGdBrd;

					IF fbSMEMA_OppFirst.udiStatus = 0 THEN
						tylocalDSSMEMA.Out.eStatus	:= Done;
					ELSIF fbSMEMA_OppFirst.udiStatus < 65534 THEN
						tylocalDSSMEMA.Out.eStatus		:= Error;

						IF fbSMEMA_OppFirst.udiStatus = 1200 THEN
							udiStatus	:= 10004;	//Standard SMEMA Transport Time Out While Transporting
						ELSIF fbSMEMA_OppFirst.udiStatus = 1201 THEN
							udiStatus	:= 10005;	//Standard SMEMA Transport Time Out After Opposite Machine Transport Finished
						ELSIF fbSMEMA_OppFirst.udiStatus = 1202 THEN
							udiStatus	:= 10006;	//Standard SMEMA Transport Time Out After Current Machine Transport Finished
						ELSIF fbSMEMA_OppFirst.udiStatus = 1203 THEN
							udiStatus	:= 10007;	//Standard SMEMA Transport Time Out After Both Machine Transport Finished And Waiting Outlet Sensor
						ELSE
							udiStatus	:= fbSMEMA_OppFirst.udiStatus;
						END_IF
					END_IF

				END_IF

			END_IF

		SMEMAActSetSig:
			IF tylocalDSSMEMA.Out.eStatus = Idle OR tylocalDSSMEMA.Out.eStatus = Busy THEN

				//Reset
				fbSMEMA_OppFirst(bEn := FALSE);
				fbSMEMA(bEn := FALSE);

				tylocalDSSMEMA.Out.bConvStart	:= FALSE;
				tylocalDSSMEMA.Out.bConvStop	:= FALSE;

				tylocalDSSMEMA.Out.bDBA	:= TRUE;
				tylocalDSSMEMA.Out.eStatus	:= Done;

			END_IF

		SMEMAActSetStatSig:
			IF tylocalDSSMEMA.Out.eStatus = Idle OR tylocalDSSMEMA.Out.eStatus = Busy THEN

				//Reset
				fbSMEMA_OppFirst(bEn := FALSE);
				fbSMEMA(bEn := FALSE);

				tylocalDSSMEMA.Out.bConvStart	:= FALSE;
				tylocalDSSMEMA.Out.bConvStop	:= FALSE;

				tylocalDSSMEMA.Out.bDBAStat	:= TRUE;
				tylocalDSSMEMA.Out.eStatus		:= Done;

			END_IF

		SMEMAActRstSig:
			IF tylocalDSSMEMA.Out.eStatus = Idle OR tylocalDSSMEMA.Out.eStatus = Busy THEN

				//Reset
				fbSMEMA_OppFirst(bEn := FALSE);
				fbSMEMA(bEn := FALSE);

				tylocalDSSMEMA.Out.bConvStart	:= FALSE;
				tylocalDSSMEMA.Out.bConvStop	:= FALSE;

				tylocalDSSMEMA.Out.bDBA	:= FALSE;
				tylocalDSSMEMA.Out.eStatus	:= Done;

			END_IF

		SMEMAActRstStatSig:
			IF tylocalDSSMEMA.Out.eStatus = Idle OR tylocalDSSMEMA.Out.eStatus = Busy THEN

				//Reset
				fbSMEMA_OppFirst(bEn := FALSE);
				fbSMEMA(bEn := FALSE);

				tylocalDSSMEMA.Out.bConvStart	:= FALSE;
				tylocalDSSMEMA.Out.bConvStop	:= FALSE;

				tylocalDSSMEMA.Out.bDBAStat	:= FALSE;
				tylocalDSSMEMA.Out.eStatus		:= Done;

			END_IF

		SMEMAActSetAllSig:
			IF tylocalDSSMEMA.Out.eStatus = Idle OR tylocalDSSMEMA.Out.eStatus = Busy THEN

				//Reset
				fbSMEMA_OppFirst(bEn := FALSE);
				fbSMEMA(bEn := FALSE);

				tylocalDSSMEMA.Out.bConvStart	:= FALSE;
				tylocalDSSMEMA.Out.bConvStop	:= FALSE;

				tylocalDSSMEMA.Out.bDBA		:= TRUE;
				tylocalDSSMEMA.Out.bDBAStat	:= TRUE;
				tylocalDSSMEMA.Out.eStatus		:= Done;

			END_IF

		SMEMAActRstAllSig:
			IF tylocalDSSMEMA.Out.eStatus = Idle OR tylocalDSSMEMA.Out.eStatus = Busy THEN

				//Reset
				fbSMEMA_OppFirst(bEn := FALSE);
				fbSMEMA(bEn := FALSE);

				tylocalDSSMEMA.Out.bConvStart	:= FALSE;
				tylocalDSSMEMA.Out.bConvStop	:= FALSE;

				tylocalDSSMEMA.Out.bDBA		:= FALSE;
				tylocalDSSMEMA.Out.bDBAStat	:= FALSE;
				tylocalDSSMEMA.Out.eStatus		:= Done;

			END_IF

	END_CASE

END_ACTION
```

#### Act_OutputConfig.st
```iecst
(** 2019-03-25 **)
ACTION Act_OutputConfig:

	(* Always Change If Project Change *)
	g_tyDSSMEMA2 := tylocalDSSMEMA.Out;

	(* Always Change If Project Change *)

END_ACTION
```

#### Cyclic.st
```iecst
(** 2019-03-29 **)
PROGRAM _CYCLIC

	IF bInitialDone = FALSE THEN
		IF g_tyStartUp.bNtSettingsLoadDone = TRUE THEN
			bInitialDone	:= TRUE;
			Act_Initial;
		END_IF

	ELSE

		Act_InputConfig;

		IF (tylocalDSSMEMA.In.bPrep = TRUE) AND (tylocalDSSMEMA.In.bEn = TRUE) AND (tylocalDSSMEMA.In.bDis = FALSE) THEN
			Act_Main;
		ELSE
			IF tylocalDSSMEMA.Out.eStat <> SMEMAActIdle THEN
				tylocalDSSMEMA.Out.eStatus	:= Done;
			ELSE
				tylocalDSSMEMA.Out.eStatus	:= Idle;
			END_IF
		END_IF

		Act_OutputConfig;
		Act_Alarm;

	END_IF

END_PROGRAM
```

#### Init.st
```iecst
(** 2019-03-25 **)
PROGRAM _INIT

	(* Always Change If Project Change *)

	//Physical Configuration
	tyParam.eSelection	:= SMEMASelIPC9851;

	//Pass Address To Global Address For External Use
	//Action, State & Status
	p_DSSMEMA2Stat		:= ADR(eStat);
	p_DSSMEMA2Status	:= ADR(eStatus);
	p_DSSMEMA2StatTxt	:= ADR(sStatTxt);

	//Alarm
	p_DSSMEMA2AlmData	:= ADR(tyAlmData);

	//Output
	p_DSSMEMA2USRdy			:= ADR(bUSRdy);
	p_DSSMEMA2USGdBrdRdy	:= ADR(bUSGdBrdRdy);
	p_DSSMEMA2DSRdy			:= ADR(bDSRdy);
	p_DSSMEMA2Transporting	:= ADR(bTransporting);
	p_DSSMEMA2ConvStart		:= ADR(bConvStart);
	p_DSSMEMA2ConvStop		:= ADR(bConvStop);
	p_DSSMEMA2DBA			:= ADR(bDBA);
	p_DSSMEMA2DBAStat		:= ADR(bDBAStat);
	p_DSSMEMA2Timer			:= ADR(bTimer);
	p_DSSMEMA2Virtual		:= ADR(bVirtual);

	//Svy Hermes
	//p_DSSMEMA2TransprtFinished	:= ADR(bDSTransportFinished);
	(* Always Change If Project Change *)

END_PROGRAM
```

### DSSMEMA3.var - Change By Project
```iecst
(*2019-03-25*)
VAR
	g_tyDSSMEMA3 : tyDSSMEMAOut1;
END_VAR
```

### Program Logical/SMEMA/DSSMEMA3 (IEC) - 1.00.0 - NtSMEMA v5.00.0

#### InputRef_Link.var
```iecst
(*2019-04-09*)
(**)
(*External Data*)
VAR
	p_bLinkOpsRun : REFERENCE TO BOOL;
END_VAR
(**)
VAR
	p_bLinkConvHvBrd : REFERENCE TO BOOL;
	p_eLinkConvDir : REFERENCE TO eConvDir;
	p_eLinkOpsTravLifPosGo : REFERENCE TO eTravLifULPos;
END_VAR
```

#### Local.var
```iecst
(*2019-04-30*)
(**)
(*Local Action, State & Status*)
VAR
	eAct : eSMEMAAction := SMEMAActIdle;
	eStat : eSMEMAAction := SMEMAActIdle;
	eStatus : eFBStatus := Idle;
	udiStatus : UDINT := 0;
	sStatTxt : STRING[200] := '';
	a_sStatText : ARRAY[0..50] OF STRING[200] := ['Idling','SMEMA Running','Turning On DBA Signal','Turning On DBA Stat Signal','Turning Off DBA Signal','Turning Off DBA Stat Signal','Turning On All DBA Signal','Turning Off All DBA Signal',43('')];
END_VAR
(**)
(*Local Alarm*)
VAR
	tyAlmData : tyAlmDat;
	a_tyAlmText : ARRAY[10000..10099] OF tyAlmTxt := [(sAlmText:='SMEMA 9851 Transport Time Out While Transporting',sRcyText:='Timeout Expired Before Operation Completed. Reset And Resume Operation.'),(sAlmText:='SMEMA 9851 Transport Time Out After Opposite Machine Transport Finished',sRcyText:='Timeout Expired Before Operation Completed. Reset And Resume Operation.'),(sAlmText:='SMEMA 9851 Transport Time Out After Current Machine Transport Finished',sRcyText:='Timeout Expired Before Operation Completed. Reset And Resume Operation.'),(sAlmText:='SMEMA 9851 Transport Time Out After Both Machine Transport Finished And Waiting Outlet Sensor',sRcyText:='Timeout Expired Before Operation Completed. Reset And Resume Operation.'),(sAlmText:='Standard SMEMA Transport Time Out While Transporting',sRcyText:='Timeout Expired Before Operation Completed. Reset And Resume Operation.'),(sAlmText:='Standard SMEMA Transport Time Out After Opposite Machine Transport Finished',sRcyText:='Timeout Expired Before Operation Completed. Reset And Resume Operation.'),(sAlmText:='Standard SMEMA Transport Time Out After Current Machine Transport Finished',sRcyText:='Timeout Expired Before Operation Completed. Reset And Resume Operation.'),(sAlmText:='Standard SMEMA Transport Time Out After Both Machine Transport Finished And Waiting Outlet Sensor',sRcyText:='Timeout Expired Before Operation Completed. Reset And Resume Operation.'),92((0))];
END_VAR
(**)
(*Local Output*)
VAR
	bUSRdy : BOOL := FALSE;
	bUSGdBrdRdy : BOOL := FALSE;
	bDSRdy : BOOL := FALSE;
	bTransporting : BOOL := FALSE;
	bConvStart : BOOL := FALSE;
	bConvStop : BOOL := FALSE;
	bDBA : BOOL := FALSE;
	bDBAStat : BOOL := FALSE;
	bTimer : BOOL;
	bVirtual : BOOL;
	bDSTransportFinished : {REDUND_UNREPLICABLE} BOOL;
END_VAR
(**)
(*Local Input*)
VAR
	udiRstErr : UDINT := 0;
	bPrep : BOOL := TRUE;
	bEn : BOOL := TRUE;
	bDis : BOOL := FALSE;
	bManual : BOOL := FALSE;
	tyParam : tySMEMAParam;
	bGdBrd : BOOL := TRUE;
	diTransferOutTO : DINT := 20000;
	bDirLToR : BOOL := FALSE;
	bRdySend : BOOL := TRUE;
	bLeftSen : BOOL := FALSE;
	bRightSen : BOOL := FALSE;
	bComplSigOn : BOOL := FALSE;
	bDSB : BOOL := FALSE;
	bTimerEnSen : BOOL;
	bTimerEnSenEdge : BOOL;
	bVirtualEn : BOOL;
	bDSBVirtual : BOOL;
	tRstDlyTm : TIME := T#500ms;
	tSigInChkTm : TIME := T#100ms;
	sProgNm : STRING[15] := 'DSSMEMA';
	bNtSettingsLoadDone : BOOL := TRUE;
END_VAR
(**)
(*Local*)
VAR
	bRstErr : BOOL;
	udiRstErrOld : UDINT;
	bInitDone : BOOL;
	bInitialDone : BOOL;
	fbTimerDlyTm : TON := (PT:=T#1s);
	fbTimeTrig : R_TRIG;
	fbSMEMA_OppFirst : fbSMEMADS_OppFirst;
	fbSMEMA : fbSMEMADS;
	fbSigInChk : fbSMEMASigInChk;
	eStatOld : eSMEMAAction := SMEMAActIdle;
	udiModuleNum : UDINT := 2801;
END_VAR
```

#### Act_Background.st
```iecst
(** 2019-01-20 **)
ACTION Act_Background:

	fbTimeTrig(CLK := p_bTimerEnSenEdge);

	IF eStat = SMEMAActRun AND (p_bTimerEnSenEdge OR p_bTimerEnSen) THEN
		IF fbTimeTrig.Q = TRUE OR p_bTimerEnSen THEN
			fbTimerDlyTm.IN	:= TRUE;
		END_IF
	ELSE
		fbTimerDlyTm.IN	:= FALSE;
	END_IF

	IF bConvStart = FALSE AND bConvStop = FALSE THEN
		fbTimerDlyTm;

		IF fbTimerDlyTm.Q = TRUE AND eStat = SMEMAActRun THEN
			bTimer		:= TRUE;
			bVirtual	:= FALSE;
		ELSIF p_bVirtualEn = TRUE THEN
			bTimer		:= FALSE;
			bVirtual	:= TRUE;
		ELSE
			bTimer		:= FALSE;
			bVirtual	:= FALSE;
		END_IF
	ELSE
		fbTimerDlyTm(IN := FALSE);
	END_IF

	IF bTimer = TRUE THEN

		fbSigInChk.bNomSig			:= bConvStart = FALSE AND bConvStop = FALSE;
		fbSigInChk.bStatSig			:= FALSE;
		fbSigInChk.bStatSigSetGd	:= FALSE;

	ELSIF bVirtual = TRUE THEN

		fbSigInChk.bNomSig			:= p_bDSBVirtual;
		fbSigInChk.bStatSig			:= FALSE;
		fbSigInChk.bStatSigSetGd	:= FALSE;

	ELSE

		fbSigInChk.bNomSig			:= p_bDSB;
		fbSigInChk.bStatSig			:= FALSE;
		fbSigInChk.bStatSigSetGd	:= FALSE;

	END_IF

	fbSigInChk;

	bDSRdy	:= fbSigInChk.bSigInValid;
//	bDSTransportFinished := bConvStart AND EDGENEG(p_bRightSen);
END_ACTION
```

#### Act_InitGlobal.st
```iecst
(** 2019-04-09 **)
ACTION Act_InitGlobal:

	(* Always Change If Project Change *)

	//Pass Data To Link
	p_bLinkOpsRun ACCESS p_OpsRun;

	p_bLinkConvHvBrd ACCESS p_PshrConvHvBrd;
	p_eLinkConvDir ACCESS p_NtParamProjConvDir;
	p_eLinkOpsTravLifPosGo ACCESS p_OpsTravLifULPosGo;

	//Pass Data To Internal Use
	p_udiRstErr ACCESS p_RstErrReset;
	p_bManual ACCESS p_UIMnlMod;
	p_bGdBrd ACCESS p_PshrConvGdBrd;
	p_bLeftSen ACCESS p_DIConvLftSen;
	p_bRightSen ACCESS p_DIConvRgtSen;
	p_bClrSen ACCESS p_DIConvClrSen;
	p_bDSB ACCESS p_USSMEMA3USB;
	p_tRstDlyTm ACCESS p_NtParamDSSMEMA3RstDlyTm;
	p_tSigInChkTm ACCESS p_NtParamDSSMEMA3SigInChkTm;
	p_sProgNm ACCESS p_NtParamDSSMEMA3ProgNm;
	p_bNtSettingsLoadDone ACCESS p_StartupNtSettingsLoadDone;

	(* Always Change If Project Change *)

END_ACTION
```

#### Act_InputConfig.st
```iecst
(** 2019-04-09 **)
ACTION Act_InputConfig:

	(* Always Change If Project Change *)

	//Pass Data To Link
	tylocalDSSMEMA.In.udiRstErr := g_tyRstErrOut.udiRstErr;
	tylocalDSSMEMA.In.bGdBrd := g_tyPshrConvGdBrd;
	tylocalDSSMEMA.In.bLeftSen := g_tyDInput.bConvLftSen;
	tylocalDSSMEMA.In.bRightSen := g_tyDInput.bConvRgtSen;
	tylocalDSSMEMA.In.bClrSen := g_tyDInput.bConvClrSen;
	tylocalDSSMEMA.In.bDSB := g_tyUSSMEMA3.bUSB;
	tylocalDSSMEMA.In.tRstDlyTm := g_tyNtParamCurr.tDSSMEMA3RstDlyTm;
	tylocalDSSMEMA.In.tSigInChkTm := g_tyNtParamCurr.tDSSMEMA3SigInChkTm;
	tylocalDSSMEMA.In.sProgNm := g_tyNtParamCurr.sDSSMEMA3ProgNm;

	(tylocalDSSMEMA.In.bRdySend	:= g_tyPshrConv.bHvBrd AND g_tyOpsTravLifUL.eTravLifULPosGo = TravLifULPosDS3;

	tylocalDSSMEMA.In.bComplSigOn	:= g_tyPshrConv.bHvBrd = FALSE AND tylocalDSSMEMA.In.bClrSen = FALSE;

	tylocalDSSMEMA.In.bDirLToR	:= g_tyNtParamCurr.eProjConvDir = ConvDirLToR OR g_tyNtParamCurr.eProjConvDir = ConvDirLToL;

	IF g_tyOps.bRun = TRUE THEN
		tylocalDSSMEMA.In.eAct := g_tyOpsTravLifULDSSMEMAAct3;
	ELSE
		tylocalDSSMEMA.In.eAct ACCESS ADR(eAct);
	END_IF

	(* Always Change If Project Change *)

END_ACTION
```

#### Act_Link.st
```iecst
(** 2019-03-29 **)
ACTION Act_Link:

	p_bRdySend	:= p_bLinkConvHvBrd AND p_eLinkOpsTravLifPosGo = TravLifULPosDS3;

	p_bComplSigOn	:= p_bLinkConvHvBrd = FALSE AND p_bClrSen = FALSE;

	p_bDirLToR	:= p_eLinkConvDir = ConvDirLToR OR p_eLinkConvDir = ConvDirLToL;

END_ACTION
```

#### Act_LinkAction.st
```iecst
(** 2019-04-09 **)
ACTION Act_LinkAction:

	IF p_bLinkOpsRun = TRUE THEN
		p_eAct ACCESS p_OpsTravLifULDSSMEMAAct3;
	ELSE
		p_eAct ACCESS ADR(eAct);
	END_IF

END_ACTION
```

#### Act_OutputConfig.st
```iecst
(** 2019-03-25 **)
ACTION Act_OutputConfig:

	(* Always Change If Project Change *)
	g_tyDSSMEMA3 := tylocalDSSMEMA.Out;

	(* Always Change If Project Change *)
END_ACTION
```

#### Init.st
```iecst
(** 2019-03-25 **)
PROGRAM _INIT

	(* Always Change If Project Change *)

	//Physical Configuration
	tyParam.eSelection	:= SMEMASelIPC9851;

	//Pass Address To Global Address For External Use
	//Action, State & Status
	p_DSSMEMA3Stat		:= ADR(eStat);
	p_DSSMEMA3Status	:= ADR(eStatus);
	p_DSSMEMA3StatTxt	:= ADR(sStatTxt);

	//Alarm
	p_DSSMEMA3AlmData	:= ADR(tyAlmData);

	//Output
	p_DSSMEMA3USRdy			:= ADR(bUSRdy);
	p_DSSMEMA3USGdBrdRdy	:= ADR(bUSGdBrdRdy);
	p_DSSMEMA3DSRdy			:= ADR(bDSRdy);
	p_DSSMEMA3Transporting	:= ADR(bTransporting);
	p_DSSMEMA3ConvStart		:= ADR(bConvStart);
	p_DSSMEMA3ConvStop		:= ADR(bConvStop);
	p_DSSMEMA3DBA			:= ADR(bDBA);
	p_DSSMEMA3DBAStat		:= ADR(bDBAStat);
	p_DSSMEMA3Timer			:= ADR(bTimer);
	p_DSSMEMA3Virtual		:= ADR(bVirtual);

	//Svy Hermes
	//p_DSSMEMA3TransprtFinished	:= ADR(bDSTransportFinished);
	(* Always Change If Project Change *)

END_PROGRAM
```

### Pneu.typ - Do Not Change!!!
```iecst
(*2018-12-11*)
(**)
(*Action*)

TYPE
	ePneuAction :
		(
		PneuActIdle,
		PneuActSetAll,
		PneuActRstAll,
		PneuActSetExt,
		PneuActSetRet,
		PneuActExt,
		PneuActRet,
		PneuActExtSenToMidSen,
		PneuActMidSenToRetSen,
		PneuActRetSenToMidSen,
		PneuActMidSenToExtSen
		);
	tyPneu : 	STRUCT
		In : tyPneuIn1;
		Out : tyPneuOut1;
	END_STRUCT;
	tyPneuIn1 : 	STRUCT
		eAct : ePneuAction := PneuActIdle; (*Enum for Actions*)
		udiRstErr : UDINT := 0; (*Reset error*)
		bPrep : BOOL := TRUE; (*Preparation*)
		bEn : BOOL := TRUE; (*Enable*)
		bDis : BOOL := FALSE; (*Disable*)
		bExtSen : BOOL := FALSE; (*Extend sensor*)
		bRetSen : BOOL := FALSE; (*Retract sensor*)
		bMidSen : BOOL := FALSE; (*Middle sensor*)
		bSafetyRelaySig : BOOL := FALSE; (*Safety Relay Signal*)
		bExtSafetySen : BOOL := TRUE; (*Extend safety sensor*)
		bRetSafetySen : BOOL := TRUE; (*Retract safety sensor*)
		bOps : BOOL := FALSE; (*Operation Mode Control*)
		bUISimu : BOOL;
		bSimu : BOOL;
		bManual : BOOL := FALSE; (*Manual mode control*)
		bTwoCtrlIn : BOOL := FALSE; (*Two way control input*)
		sProgNm : STRING[15] := 'Pneu2Sen'; (*Program title name*)
		tExtTO : TIME := T#20s; (*Extend timer*)
		tRetTO : TIME := T#20s; (*Retract timer*)
		bNtSettingsLoadDone : BOOL := TRUE; (*Nutek settings load done*)
		tExtDlyTm : TIME := T#1s; (*Extend delay time*)
		tRetDlyTm : TIME := T#1s; (*Retract delay time*)
		ePneuSel : ePneuSel1;
		bLinkDIConvClrSen : BOOL;
		bConvPusherReachedRetSlw : BOOL;
		bLinkDIPusherRetRS : BOOL;
		eLinkLifterBtmStat : eLifterAction;
		eLinkLifterBtmStatus : eFBStatus;
		eLinkLifter2Stat : eLifterAction;
		eLinkLifter2Status : eFBStatus;
		bNtParamProjLifter2Prep : BOOL;
		bMagRcpCurrRcpSBarDisabled : REFERENCE TO BOOL;
	END_STRUCT;
	tyPneuOut1 : 	STRUCT
		bExtCtrl : BOOL; (*Extend control*)
		bRetCtrl : BOOL; (*Retract control*)
		bExtended : BOOL;
		bRetracted : BOOL;
		bTwoCtrlOut : BOOL := FALSE; (*Two way control output*)
		eStat : ePneuAction := PneuActIdle; (*Enum for Actions.*)
		eStatus : eFBStatus := Idle; (*Status*)
		sStatTxt : STRING[200] := ''; (*Status/ alarm message*)
		tyAlmData : tyAlmDat; (*Alarm data structure type.*)
	END_STRUCT;
	ePneuSel1 :
		(
		PneuNoSen := 0,
		PneuExtSen := 1,
		PneuRetSen := 2,
		Pneu2Sen := 3,
		Pneu3Sen := 4
		);
END_TYPE
```

### Pneu.var - Change By Project
```iecst
VAR
	g_tyPneuInShutter : tyPneuOut1; (*OutletShutter*)
	g_tyPneuOutShutter : tyPneuOut1; (*OutletShutter*)
	g_tyPneuOutShutter2 : tyPneuOut1; (*OutletShutter*)
	g_tyPneuOutShutter3 : tyPneuOut1; (*OutletShutter*)
	g_tyPneuStopperA : tyPneuOut1;
	g_tyPneuStopperB : tyPneuOut1;
	g_tyPneuStopperC : tyPneuOut1;
	g_tyPneuSelClamp1 : tyPneuOut1;
	g_tyPneuSelClamp2 : tyPneuOut1;
	g_tyPneuSelClamp3 : tyPneuOut1;
	g_tyPneuMag1SafetyBar : tyPneuOut1;
	g_tyPneuMag2SafetyBar : tyPneuOut1;
	g_tyPneuMag3SafetyBar : tyPneuOut1;
	g_tyPneuMag1AWEngage : tyPneuOut1;
	g_tyPneuMag2AWEngage : tyPneuOut1;
	g_tyPneuMag3AWEngage : tyPneuOut1;
END_VAR
```

### Program Logical/Pneu/PneuInShutter (IEC) - 1.00.0 - NtPneu v5.00.0

#### Act_InputConfig.st
```iecst
(** 2019-04-09 **)
ACTION Act_InputConfig:

// Input: Assign From Machine Parameter/Nutek Parameter/Digital input&output/Required Triggering Flags From Other Packages
	//Pass Data To Link
	tylocalPneu.In.bSafetyRelaySig 	 	 := g_tyDInput.bSafetyRlySig;
	tylocalPneu.In.udiRstErr		 	 := g_tyRstErrOut.udiRstErr;
	tylocalPneu.In.bPrep			  	 := g_tyNtParamCurr.bProjInletShutPrep;
	tylocalPneu.In.bDis			  	 	 := g_tyMcParamCurr.bInShutterDis;
	tylocalPneu.In.bUISimu		  	 	 := g_tyUIOut.bSimuMod;
	tylocalPneu.In.bManual		  	 	 := g_tyUIOut.bUIManualMod;
	tylocalPneu.In.bTwoCtrlIn		 	 := g_tyNtParamCurr.bInShutterTwoCtrlIn;
	tylocalPneu.In.sProgNm			 	 := g_tyNtParamCurr.sInShutterProgNm;
	tylocalPneu.In.bExtSen			 	 := g_tyDInput.bInShutterCloseRS;
	tylocalPneu.In.bRetSen			 	 := g_tyDInput.bInShutterOpenRS;

	tylocalPneu.In.tExtTO			 	 := g_tyNtParamCurr.tInShutterExtTO;
	tylocalPneu.In.tRetTO		 	     := g_tyNtParamCurr.tInShutterRetTO ;
	tylocalPneu.In.ePneuSel				 := Pneu2Sen; //Pneumatic With 2 Sensors

	//Link bPrep, bEn & bDis
	IF g_tyStartUp.bRun THEN
		tylocalPneu.In.bDis	 := p_bLinkMcParamInShutDis AND g_tyOpsTravLifUL.bInitDone;
	ELSE
		tylocalPneu.In.bDis	 := FALSE;
	END_IF

	IF g_tyOps.bRun = TRUE THEN
		tylocalPneu.In.eAct := g_tyOpsTravLifUL.eInletPneuAct;
	ELSIF tylocalPneu.In.bManual = TRUE OR tylocalPneu.In.bUISimu THEN
		tylocalPneu.In.eAct := g_tyUIOut.eMnlAct.eInShutterAct;
	ELSE
		tylocalPneu.In.eAct := eAct;
	END_IF

	(* Always Change If Project Change *)

END_ACTION
```

#### Act_Main.st
```iecst
ACTION Act_Main:

	IF tylocalPneu.In.bSafetyRelaySig = FALSE OR EDGEPOS(tylocalPneu.Out.eStatus = Error) THEN
		tylocalPneu.Out.bExtCtrl 	:= FALSE;
		tylocalPneu.Out.bRetCtrl 	:= FALSE;
		tylocalPneu.Out.bExtended	:= FALSE;
		tylocalPneu.Out.bRetracted  := FALSE;
	END_IF

	//Execution Action
	IF tylocalPneu.Out.eStatus <> Error THEN
		tylocalPneu.Out.eStat := tylocalPneu.In.eAct;
	END_IF

	//Transition State
	IF eStatOld <> tylocalPneu.Out.eStat THEN

		fbPneuNoSenExt(bEn := FALSE);
		fbPneuNoSenRet(bEn := FALSE);

		fbPneu2SenExt(bEn := FALSE);
		fbPneu2SenRet(bEn := FALSE);

		eStatOld	:= tylocalPneu.Out.eStat;

		tylocalPneu.Out.eStatus		:= Busy;
	END_IF

	//Main
	CASE tylocalPneu.Out.eStat OF

		PneuActIdle:
			tylocalPneu.Out.eStatus	:= Idle;

		PneuActSetAll:
			IF tylocalPneu.Out.eStatus = Idle OR tylocalPneu.Out.eStatus = Busy THEN

				fbPneuNoSenExt(bEn := FALSE);
				fbPneuNoSenRet(bEn := FALSE);

				fbPneu2SenExt(bEn := FALSE);
				fbPneu2SenRet(bEn := FALSE);

				tylocalPneu.Out.bExtCtrl	:= TRUE;
				tylocalPneu.Out.bRetCtrl	:= TRUE;

				tylocalPneu.Out.bExtended	:= FALSE;
				tylocalPneu.Out.bRetracted	:= FALSE;

				tylocalPneu.Out.eStatus	:= Done;

			END_IF

		PneuActRstAll:
			IF tylocalPneu.Out.eStatus = Idle OR tylocalPneu.Out.eStatus = Busy THEN

				fbPneuNoSenExt(bEn := FALSE);
				fbPneuNoSenRet(bEn := FALSE);

				fbPneu2SenExt(bEn := FALSE);
				fbPneu2SenRet(bEn := FALSE);

				tylocalPneu.Out.bExtCtrl	:= FALSE;
				tylocalPneu.Out.bRetCtrl	:= FALSE;

				tylocalPneu.Out.bExtended	:= FALSE;
				tylocalPneu.Out.bRetracted	:= FALSE;

				tylocalPneu.Out.eStatus	:= Done;

			END_IF

		PneuActSetExt:
			IF tylocalPneu.Out.eStatus = Idle OR tylocalPneu.Out.eStatus = Busy THEN

				fbPneuNoSenExt(bEn := FALSE);
				fbPneuNoSenRet(bEn := FALSE);

				fbPneu2SenExt(bEn := FALSE);
				fbPneu2SenRet(bEn := FALSE);

				tylocalPneu.Out.bExtCtrl	:= TRUE;
				tylocalPneu.Out.bRetCtrl	:= FALSE;

				tylocalPneu.Out.bExtended	:= TRUE;
				tylocalPneu.Out.bRetracted	:= FALSE;

				tylocalPneu.Out.eStatus	:= Done;

			END_IF

		PneuActSetRet:
			IF tylocalPneu.Out.eStatus = Idle OR tylocalPneu.Out.eStatus = Busy THEN

				//Reset
				fbPneuNoSenExt(bEn := FALSE);
				fbPneuNoSenRet(bEn := FALSE);

				fbPneu2SenExt(bEn := FALSE);
				fbPneu2SenRet(bEn := FALSE);

				tylocalPneu.Out.bExtCtrl	:= FALSE;
				tylocalPneu.Out.bRetCtrl	:= TRUE;

				tylocalPneu.Out.bExtended	:= FALSE;
				tylocalPneu.Out.bRetracted	:= TRUE;

				tylocalPneu.Out.eStatus	:= Done;

			END_IF

		PneuActExt:
			IF tylocalPneu.Out.eStatus = Idle OR tylocalPneu.Out.eStatus = Busy THEN

				tylocalPneu.Out.eStatus	:= Busy;

				tylocalPneu.Out.bExtCtrl	:= TRUE;
				tylocalPneu.Out.bRetCtrl	:= FALSE;

				CASE tylocalPneu.In.ePneuSel OF

					PneuNoSen: //Pneumatic Without Sen // 0
						fbPneuNoSenExt.bExtSafety	:= tylocalPneu.In.bExtSafetySen;
						fbPneuNoSenExt.tDlyTm		:= tylocalPneu.In.tExtDlyTm;
						fbPneuNoSenExt(bEn := TRUE);
					Pneu2Sen: //Pneumatic With 2 Sen // 3
						fbPneu2SenExt.bExtSen   	:= tylocalPneu.In.bExtSen;
						fbPneu2SenExt.bRetSen   	:= tylocalPneu.In.bRetSen;
						fbPneu2SenExt.bExtSafety	:= tylocalPneu.In.bExtSafetySen;
						fbPneu2SenExt.tTimeOut		:= tylocalPneu.In.tExtTO;
						fbPneu2SenExt(bEn := TRUE);
				END_CASE

				IF fbPneuNoSenExt.udiStatus = 0 OR
					fbPneu2SenExt.udiStatus = 0 THEN

					tylocalPneu.Out.bExtended	:= TRUE;
					tylocalPneu.Out.bRetracted	:= FALSE;
					tylocalPneu.Out.eStatus		:= Done;

				ELSIF (fbPneuNoSenExt.udiStatus > 0 AND fbPneuNoSenExt.udiStatus < 65534) OR
					(fbPneu2SenExt.udiStatus > 0 AND fbPneu2SenExt.udiStatus < 65534) THEN

					IF tylocalPneu.In.bTwoCtrlIn = TRUE THEN

						tylocalPneu.Out.bExtCtrl	:= FALSE;
						tylocalPneu.Out.bRetCtrl	:= FALSE;

					ELSE
						tylocalPneu.Out.bExtCtrl	:= FALSE;
						tylocalPneu.Out.bRetCtrl	:= TRUE;

					END_IF

					tylocalPneu.Out.bExtended	:= FALSE;
					tylocalPneu.Out.bRetracted	:= FALSE;

					tylocalPneu.Out.eStatus		:= Error;

					IF fbPneuNoSenExt.udiStatus = 1507 OR fbPneu2SenExt.udiStatus  = 1507 THEN
						udiStatus	:= 2401; //Safety Check Error While Extending
					ELSIF fbPneu2SenExt.udiStatus = 1503 THEN
						udiStatus	:= 2552;	//Extend Sensor On Checking Time Out While Extending
					ELSIF fbPneu2SenExt.udiStatus = 1506 THEN
						udiStatus	:= 2553; //Retract Sensor Off Checking Time Out While Extending
					ELSE
						IF tylocalPneu.In.ePneuSel = PneuNoSen THEN
							udiStatus	:= fbPneuNoSenExt.udiStatus;
						ELSE
							udiStatus	:= fbPneu2SenExt.udiStatus;
						END_IF
					END_IF
				END_IF

			END_IF

		PneuActRet:
			IF tylocalPneu.Out.eStatus = Idle OR tylocalPneu.Out.eStatus = Busy THEN

				tylocalPneu.Out.eStatus	:= Busy;

				tylocalPneu.Out.bExtCtrl	:= FALSE;
				tylocalPneu.Out.bRetCtrl	:= TRUE;

				CASE tylocalPneu.In.ePneuSel OF

					PneuNoSen: //Pneumatic Without Sen // 0
						fbPneuNoSenRet.bRetSafety	:= tylocalPneu.In.bRetSafetySen;
						fbPneuNoSenRet.tDlyTm		:= tylocalPneu.In.tRetDlyTm;
						fbPneuNoSenRet(bEn := TRUE);
					Pneu2Sen: //Pneumatic With 2 Sen // 3
						fbPneu2SenRet.bExtSen   	:= tylocalPneu.In.bExtSen;
						fbPneu2SenRet.bRetSen   	:= tylocalPneu.In.bRetSen;
						fbPneu2SenRet.bRetSafety	:= tylocalPneu.In.bRetSafetySen;
						fbPneu2SenRet.tTimeOut		:= tylocalPneu.In.tRetTO;
						fbPneu2SenRet(bEn := TRUE);
				END_CASE

				IF fbPneuNoSenRet.udiStatus = 0 OR
					fbPneu2SenRet.udiStatus = 0 THEN

					tylocalPneu.Out.bExtended	:= FALSE;
					tylocalPneu.Out.bRetracted	:= TRUE;
					tylocalPneu.Out.eStatus		:= Done;

				ELSIF (fbPneuNoSenRet.udiStatus > 0 AND fbPneuNoSenRet.udiStatus < 65534) OR
					(fbPneu2SenRet.udiStatus > 0 AND fbPneu2SenRet.udiStatus < 65534) THEN

					IF tylocalPneu.In.bTwoCtrlIn = TRUE THEN
						tylocalPneu.Out.bExtCtrl	:= FALSE;
						tylocalPneu.Out.bRetCtrl	:= FALSE;
					ELSE
						tylocalPneu.Out.bExtCtrl	:= TRUE;
						tylocalPneu.Out.bRetCtrl	:= FALSE;
					END_IF

					tylocalPneu.Out.bExtended	:= FALSE;
					tylocalPneu.Out.bRetracted	:= FALSE;

					tylocalPneu.Out.eStatus		:= Error;

					IF fbPneuNoSenRet.udiStatus = 1508 OR fbPneu2SenRet.udiStatus = 1508 THEN
						udiStatus	:= 2404;	//Safety Check Error While Retracting
					ELSIF fbPneu2SenRet.udiStatus = 1505 THEN
						udiStatus	:= 2555;	//Retract Sensor On Checking Time Out While Retracting
					ELSIF fbPneu2SenRet.udiStatus = 1504 THEN
						udiStatus	:= 2556;    //Extend Sensor Off Checking Time Out While Retracting
					ELSE
						IF tylocalPneu.In.ePneuSel = PneuNoSen THEN
							udiStatus	:= fbPneuNoSenRet.udiStatus;
						ELSE
							udiStatus	:= fbPneu2SenRet.udiStatus;
						END_IF
					END_IF
				END_IF

			END_IF

		ELSE
			IF tylocalPneu.Out.eStatus = Idle OR tylocalPneu.Out.eStatus = Busy THEN
				tylocalPneu.Out.eStatus	:= Done;
			END_IF

	END_CASE

	//background
	IF tylocalPneu.In.ePneuSel = Pneu2Sen THEN
		IF tylocalPneu.In.bExtSen = FALSE THEN
			tylocalPneu.Out.bExtended	:= FALSE;
		END_IF

		IF tylocalPneu.In.bRetSen = FALSE THEN
			tylocalPneu.Out.bRetracted	:= FALSE;
		END_IF
	END_IF

END_ACTION
```

#### Act_OutputConfig.st
```iecst
ACTION Act_OutputConfig:

// Output: Assign To Global For Independent Package Usage

 g_tyPneuInShutter := tylocalPneu.Out; // Change the Global Naming According to the Physical Hardware Module

END_ACTION
```

#### Cyclic.st
```iecst
(** 2019-03-29 **)
PROGRAM _CYCLIC

	IF bInitialDone = FALSE THEN
		IF 	g_tyStartUp.bNtSettingsLoadDone = TRUE THEN
			bInitialDone	:= TRUE;
			Act_Initial;
		END_IF
	ELSE

		Act_InputConfig;

		IF (tylocalPneu.In.bPrep = TRUE) AND (tylocalPneu.In.bEn = TRUE) AND (tylocalPneu.In.bDis = FALSE) THEN
			Act_Main;
		ELSE
			IF tylocalPneu.Out.eStat <> PneuActIdle THEN
				IF eStat = PneuActSetExt OR eStat = PneuActExt THEN
					tylocalPneu.Out.bExtended	:= TRUE;
					tylocalPneu.Out.bRetracted	:= FALSE;
				ELSIF eStat = PneuActSetRet OR eStat = PneuActRet THEN
					tylocalPneu.Out.bExtended	:= FALSE;
					tylocalPneu.Out.bRetracted	:= TRUE;
				END_IF
				tylocalPneu.Out.eStatus	:= Done;
			ELSE
				tylocalPneu.Out.eStatus	:= Idle;
			END_IF
		END_IF

		Act_OutputConfig;

		Act_Alarm;

	END_IF

END_PROGRAM
```

### Program Logical/Pneu/PneuOutShutter (IEC) - 1.00.0 - NtPneu v5.00.0

#### Act_Initial.st
```iecst
ACTION Act_Initial:

	fbPneuNoSenExt(bEn := FALSE);
	fbPneuNoSenRet(bEn := FALSE);
	fbPneu2SenExt(bEn := FALSE);
	fbPneu2SenRet(bEn := FALSE);

END_ACTION
```
